// TwinCAT 3 PLC project DrivePLC
// ProgramVersion: 3.1.4020.4
// libraries:
//   Tc2_MC2, * (Beckhoff Automation GmbH)
//   Tc2_MC2_Camming, * (Beckhoff Automation GmbH)
//   Tc2_NC, * (Beckhoff Automation GmbH)
//   Tc2_Standard, * (Beckhoff Automation GmbH)
//   Tc2_System, * (Beckhoff Automation GmbH)
//   Tc3_MC2_AdvancedHoming, * (Beckhoff Automation GmbH)
//   Tc3_Module, * (Beckhoff Automation GmbH)
//   VisuDialogs, * (System)
// project tree:
//   DUTs/ ST_AxisControl.TcDUT, eLimitCoupling.TcDUT, eMcCommand.TcDUT, eRWParameter.TcDUT, ST_MasterAxis.TcDUT, ST_MasterCoupling.TcDUT, ST_SimulateStage.TcDUT
//   / GlobalTextList.TcGTLO, PlcTask.TcTTO, Visualization Manager.TcVMO (not stored)
//   GVLs/ GVL.TcGVL, Limits.TcGVL
//   POUs/ FB_AxisDrive.TcPOU, MAIN.TcPOU
//   VISUs/COMMAND VISUS/ Gearing.TcVIS, Parameters.TcVIS, Homing.TcVIS, AxisSimulation.TcVIS
//   VISUs/ Main.TcVIS
//   VISUs/Panels/ ButtonStates.TcTLO, CommandList.TcTLO, ImagePool.TcIPO (not stored), IO.TcVIS, SlitSet.TcVIS, Visualization.TcVIS
//   VISUs/Panels/Command VISUs/ AxisSimulation.TcVIS, Gearing.TcVIS, Homing.TcVIS, Parameters.TcVIS
// real-time tasks:
//   TASK PlcTask: cycle T#10ms, priority 20, ADS port 350
//   TASK VISU_TASK: cycle T#200000us, priority 30, ADS port 351
// motion (NC):
//   TASK NC-Task 1 SAF: cycle T#2ms, priority 4, ADS port 501
//   TASK NC-Task 1 SVB: cycle T#10ms, priority 8, ADS port 511
//   AXIS NORTH (id 1)
//     General: UnitName=Degree
//     Dynamic: AccelerationMaximum=1500, Acceleration=119.286, Deceleration=119.286, Jerk=424.749
//     Velo: SlowManual=10, FastManual=50, Maximum=50
//     OtherSettings: AllowMotionCmdToSlave=true
//     encoder EncType=1
//     drive DrvType=5
//       Analog: ScaleFactorActTorque=0.1
//       TimeComp: TaskDelayCycles=1
//     controller CtrType=1
//       CtrPara: PriorControlFactor=1
//         Observer: BandWidth=20
//   AXIS SOUTH (id 2)
//     General: UnitName=Degree
//     Dynamic: AccelerationMaximum=1500
//     Velo: SlowManual=10, FastManual=50, Maximum=50
//     OtherSettings: AllowMotionCmdToSlave=true
//     encoder EncType=1
//       EncPara: ScaleFactorNumerator=0.09, Inverse=true
//         SoftEndMaxControl: Range=360
//         Inc: RefSearchInverse=true, RefSyncInverse=false, RefSoftSyncMask=#x0000ffff
//     drive DrvType=5
//       Analog: ScaleFactorActTorque=0.1
//       TimeComp: TaskDelayCycles=1
//     controller CtrType=1
//       CtrPara: PriorControlFactor=1
//         Observer: BandWidth=20
//   AXIS EAST (id 3)
//     General: UnitName=Degree
//     Dynamic: AccelerationMaximum=1500
//     Velo: SlowManual=10, FastManual=50, Maximum=50
//     OtherSettings: AllowMotionCmdToSlave=true
//     encoder EncType=1
//       SoftEndMinControl: Range=-180
//       SoftEndMaxControl: Range=180
//     drive DrvType=5
//       Analog: ScaleFactorActTorque=0.1
//       TimeComp: TaskDelayCycles=1
//     controller CtrType=1
//       CtrPara: PriorControlFactor=1
//         Observer: BandWidth=20
//   AXIS WEST (id 4)
//     Dynamic: AccelerationMaximum=1500
//     Velo: SlowManual=10, FastManual=50, Maximum=50
//     OtherSettings: AllowMotionCmdToSlave=true
//     encoder EncType=1
//       SoftEndMinControl: Range=-180
//       SoftEndMaxControl: Range=180
//     drive DrvType=5
//       Analog: ScaleFactorActTorque=0.1
//       TimeComp: TaskDelayCycles=1
//     controller CtrType=1
//       CtrPara: PriorControlFactor=1
//         Observer: BandWidth=20
//   AXIS VG (id 5)
//     Dynamic: AccelerationMaximum=1500
//     Velo: SlowManual=10, FastManual=50, Maximum=50
//     OtherSettings: AllowMotionCmdToSlave=true
//     encoder EncType=1
//       Inc: RefSoftSyncMask=#x0000ffff
//     drive DrvType=5
//       Analog: ScaleFactorActTorque=0.1
//       TimeComp: TaskDelayCycles=1
//     controller CtrType=1
//       CtrPara: PriorControlFactor=1
//         Observer: BandWidth=20
//   AXIS VC (id 6)
//     Dynamic: AccelerationMaximum=1500
//     Velo: SlowManual=10, FastManual=50, Maximum=50
//     OtherSettings: AllowMotionCmdToSlave=true
//     encoder EncType=1
//     drive DrvType=5
//       Analog: ScaleFactorActTorque=0.1
//       TimeComp: TaskDelayCycles=1
//     controller CtrType=1
//       CtrPara: PriorControlFactor=1
//         Observer: BandWidth=20
//   AXIS HG (id 7)
//     Dynamic: AccelerationMaximum=1500
//     Velo: SlowManual=10, FastManual=50, Maximum=50
//     OtherSettings: AllowMotionCmdToSlave=true
//     encoder EncType=1
//     drive DrvType=5
//       Analog: ScaleFactorActTorque=0.1
//       TimeComp: TaskDelayCycles=1
//     controller CtrType=1
//       CtrPara: PriorControlFactor=1
//         Observer: BandWidth=20
//   AXIS HC (id 8)
//     Dynamic: AccelerationMaximum=1500
//     Velo: SlowManual=10, FastManual=50, Maximum=50
//     OtherSettings: AllowMotionCmdToSlave=true
//     encoder EncType=1
//     drive DrvType=5
//       Analog: ScaleFactorActTorque=0.1
//       TimeComp: TaskDelayCycles=1
//     controller CtrType=1
//       CtrPara: PriorControlFactor=1
//         Observer: BandWidth=20
// variable links:
//   DrivePLC Instance <-> NC-Task 1 SAF/Axes/EAST
//     PlcTask Inputs/GVL.axes[3].Axis.NcToPlc <-> Outputs/ToPlc
//     PlcTask Outputs/GVL.axes[3].Axis.PlcToNc <-> Inputs/FromPlc
//   DrivePLC Instance <-> NC-Task 1 SAF/Axes/HC
//     PlcTask Inputs/GVL.axes[8].Axis.NcToPlc <-> Outputs/ToPlc
//     PlcTask Outputs/GVL.axes[8].Axis.PlcToNc <-> Inputs/FromPlc
//   DrivePLC Instance <-> NC-Task 1 SAF/Axes/HG
//     PlcTask Inputs/GVL.axes[7].Axis.NcToPlc <-> Outputs/ToPlc
//     PlcTask Outputs/GVL.axes[7].Axis.PlcToNc <-> Inputs/FromPlc
//   DrivePLC Instance <-> NC-Task 1 SAF/Axes/NORTH
//     PlcTask Inputs/GVL.axes[1].Axis.NcToPlc <-> Outputs/ToPlc
//     PlcTask Outputs/GVL.axes[1].Axis.PlcToNc <-> Inputs/FromPlc
//   DrivePLC Instance <-> NC-Task 1 SAF/Axes/SOUTH
//     PlcTask Inputs/GVL.axes[2].Axis.NcToPlc <-> Outputs/ToPlc
//     PlcTask Outputs/GVL.axes[2].Axis.PlcToNc <-> Inputs/FromPlc
//   DrivePLC Instance <-> NC-Task 1 SAF/Axes/VC
//     PlcTask Inputs/GVL.axes[6].Axis.NcToPlc <-> Outputs/ToPlc
//     PlcTask Outputs/GVL.axes[6].Axis.PlcToNc <-> Inputs/FromPlc
//   DrivePLC Instance <-> NC-Task 1 SAF/Axes/VG
//     PlcTask Inputs/GVL.axes[5].Axis.NcToPlc <-> Outputs/ToPlc
//     PlcTask Outputs/GVL.axes[5].Axis.PlcToNc <-> Inputs/FromPlc
//   DrivePLC Instance <-> NC-Task 1 SAF/Axes/WEST
//     PlcTask Inputs/GVL.axes[4].Axis.NcToPlc <-> Outputs/ToPlc
//     PlcTask Outputs/GVL.axes[4].Axis.PlcToNc <-> Inputs/FromPlc

CONFIGURATION DrivePLC
    RESOURCE PLC ON TwinCAT3
        TASK PlcTask(INTERVAL := T#10ms, PRIORITY := 20);
        PROGRAM MAIN WITH PlcTask : MAIN;
    END_RESOURCE
END_CONFIGURATION

// ---- DUTs/ST_AxisControl.TcDUT
TYPE ST_AxisControl :
STRUCT
	//OPC UA functionality not implemented yet
	(*For a list of parameters required to operate each motion control funciton block
	see the DUT eMcCommand*)
	
	bExecute			:	BOOL;			//Rising edge to execute command
	bReset				:	BOOL;			//Reset axis signal, must be combined with other signals
	eCommand			:	eMcCommand;		//Motion command for axis
	bEnable				: 	BOOL;			//Controller enable
	fOverride			:	LREAL;			//Controller override %
	fVelocity			:	LREAL;			//Velocity must be specified, no default used
	fAcceleration		:	LREAL;			//Not all FBs use, need to change this, 0 is NC default
	fDeceleration		:	LREAL;			//Not all FBs use, need to change this, 0 is NC default
	fDistance			:	LREAL;			//Used for relative positioning
	fPosition			:	LREAL;			//Used for absolute positioning	
	bJogForward			:	BOOL;			//Jog forward
	bJogBackward		:	BOOL;			//Jog backward
	
	bInput				:	BOOL;			//Generic input that is utilised to control some functionality
	
	bSoftLimPosEn		:	BOOL;			//Enable/disable positive direction software limit
	bSoftLimNegEn		:	BOOL;			//Enable/disable negative direction software limit
	bPosLagEn			:	BOOL;			//Enable/disable position lag
	
	//Gearing parameters
	masterAxis			:	UINT:=1;						//Axes[ ] index for master		- GearIn
	fGearRatioNum		:	LREAL;							//GearIn ratio numerator
	iGearRatioDen		:	UINT;							//GearIn ratio denominator
	masterAxes			:	ARRAY[1..4] OF ST_MasterAxis;	//ST to hold index and ratio for masters 	- GearInMultiMaster
	
	//NC Parameters	
	iParameterIndex		:	INT;					//Index for checking parameters
	fParameterValue		:	LREAL;					//Holder for assigning new values
	fParameters			:	ARRAY [1..17] OF LREAL;	//Array to hold NC parameters
	
	//MISC
	sAxisName			:	STRING;					//User set name string for axis
	sAxisDesc			:	STRING;					//User set description string for axis
	
	//Outputs
	bFwEnabled			:	BOOL;					//Positive movement of axis is enabled/disabled
	bBwEnabled			:	BOOL;					//Negative movement of axis is enabled/disabled
	bAxisReady			:	BOOL;					//Output of McPower block	
	bError				:	BOOL;					//Motion function block has produced error (NC drive not necessarily in error state)
	iErrorID			:	UDINT;					//Motion function block errorID				
	bBusy				:	BOOL;					//Axis busy
	bMoving				:	BOOL;					//Axis moving					
	bDone				:	BOOL;					//Last function block executed successfully			
	
	iAxisState			:	UINT;					//PLC Open NC statemachine, int assigned to individual NC bool state outputs
	(*	100 - Disabled
		200 - Standstill
		300 - Homing
		400 - Discrete Motion
		500 - Synchronized Motion
		600 - Continuous Motion
		700 - Stopping
		999 - Error
	*)
	
	buffer				:	MC_BufferMode;							//Placeholder - Not currently used
	
	//Homing
	fHomeVelocity		:	LREAL	:=1;							//Homing routine velocity 							- initialised for testing purposes
	fHomeTorque			:	LREAL;									//Homing torque limit (not all drives support this)
	fHomePosition		:	LREAL;									//Position set at NC when homing step finished
	fHomeDistance		:	LREAL;									//Relative distance to move after homing
	tHomeTimeLimit		:	TIME:=T#60S;							//Homing timeout limit, FB errors is exceeded 		- initialised for testing purposes
	fHomeDistanceLimit	:	LREAL:=2000;							//Homing distance limit, FB errors if exceeded 		- initialised for testing purposes
	
	MCHomeDirection		:	MC_Home_Direction:=	mcSwitchPositive;	//init for testing purposes
	(*	Direction to begin homing. Not all are compatible with every advanced homing step
		mcPositiveDirection	-	always start positive
		mcNegativeDirection	-	always start negative
		mcSwitchPositive	-	start positive unless already on the switch
		mcSwitchNegative	-	start negative unless already on the switch
		
	*)
	

	MCSwitchMode		:	MC_Switch_Mode:= mcRisingEdge;			//init for testing purposes
	(* Switch detection behaviour, I am not entirely convinced these are all working as they are meant to, further work required. Not all detection methods work with every 
	step either so they have to be updated.
		mcOn
		mcOff
		mcRisingEdge
		mcFallingEdge
		mcEdgeSwitchPositive
		mcEdgeSwitchNegative
		mcRisingEdgeInverse
		mcFallingEdgeInverse	
	*)

	MCSignalRef			:	MC_Ref_Signal_Ref;						//In structure for testing purposes so I can simulate level of signal without hardware
	(*Further investigation required on how exactly this MCSignalRef works, it seems to contain signalsource, touch probe and level signals,
	my current understanding is that with physical hardware connected the MCSignalRef signal source should default to the NC hardware so nothing has to be linked
	for the encoder index, however the source may need to be changed for the absSwitch homing which would just require an additional line of code in the driveFB step command
	I also do not have any bool available for linking an absolute switch to an axis at the moment

		SignalSource : E_SignalSource := SignalSource_Default;
		TouchProbe : E_TouchProbe := PlcEvent;
		Level : BOOL;

	*)

	// Data for EPICS from the axis ref
	fActPosition   			: LREAL;
	fActVelocity  		 	: LREAL;
	bNegativeDirection 		: BOOL;
	bPositiveDirection		: BOOL;
	bCalibrated 			: BOOL;
	
	Axis				:	AXIS_REF;		(*~ (OPC: 0 : available for OPC-clients) *)

END_STRUCT
END_TYPE

// ---- DUTs/eLimitCoupling.TcDUT
{attribute 'qualified_only'}
{attribute 'strict'}
(*
	Structure used to couple limit switches of slaves to master axes
*)
TYPE eLimitCoupling :
(
	None,
	FwSw,
	BwSw
);
END_TYPE

// ---- DUTs/eMcCommand.TcDUT
{attribute 'qualified_only'}
{attribute 'strict'}
TYPE eMcCommand :
(
	(*
		Only those with listed inputs have been implemented, the rest are placeholders to be added 
		To utilise a listed command you must give the ST_AxisControl the listed inputs, the drive function block will latch on a command until it is complete or errors 
		and the bExecute signal will be automatically set FALSE on every cycle
	*)
	
	Idle,					//Internal idle command, 	Inputs	:	NONE
	Reset,					//Reset NC axis,			Inputs	:	bReset
	ReadAxisError,
	WriteParameter,			//Write to NC parameters,	Inputs	:	bExecute	iParameterIndex		fParameterValue
	WriteBoolParameter,		//Write to NC parameters,	Inputs	:	bExecute	iParameterIndex		bInput

	ReadActualPosition,
	ReadActualVelocity,

	
	SetPosition,			//Set NC axis position,		Inputs	:	bExecute	fPosition			
	SetOverride,
	TouchProbe,
	
	AbortTrigger,
	AbortSuperposition,
	CamTableSelect,
	
	Home,
	Jog,					//Jog the axis,				Inputs	:	bJogForward		bJogBackward
	Stop,					//Stop axis motion,			Inputs	:	bExecute	fDeceleration
	Halt,
	MoveAbsolute,			//Absolute move,			Inputs	:	bExecute	fPosition	fVelocity	fAcceleration	fDeceleration
	MoveRelative,			//Relative move,			Inputs	:	bExecute	fDistance	fVelocity	fAcceleration	fDeceleration
	MoveAdditive,
	MoveSuperimposed,
	MoveVelocity,			//Velocity move,			Inputs	:	bExecute	fVelocity	fAcceleration	fDeceleration
	MoveContinuousAbs,
	MoveContinuousRel,
	MoveModulo,
	
	GearIn,					//Single master gear in,	Inputs	:	bExecute	fGearRatioNum	iGearRatioDen	masterAxis
	GearInDyn,
	GearInMultiMaster,		//Multi master gear in,		Inputs	:	bExecute	fGearRatio1		fGearRatio2		fGearRatio3		fGearRatio4		masterAxis1		masterAxis2		masterAxis3		masterAxis4
	GearOut,				//Release gearing,			Inputs	:	bExecute	
	HaltPhasing,
	PhasingAbsolute,
	PhasingRelative,
	CamIn,
	CamOut,
	CamScaling,
	CamAdd,
	CamExchange,
	CamInV2,
	CamRemove,
	CamScalingV2,
	
	//HOMING		Those marked with * have had values initialised and don't need to be input (but can be)
	HomeFinish,				//Finish homing routin,		Inputs	:	bExecute	fHomeDistance	fHomeVelocity
	HomeDirect,
	HomeAbort,
	HomeStepAbsoluteSwitch,	//Homing step,				Inputs	:	bExecute	MCHomeDirection*	mcSwitchMode*	mcSignalRef*	fHomeVelocity*	fHomeTorque		fHomePosition	tHomeTimeLimit*		fHomeDistanceLimit*		buffer*
	HomeStepBlock,
	HomeStepBlockLagBased,
	HomeStepLimitSwitch,
	HomeStepReferencePulse
	
);
END_TYPE

// ---- DUTs/eRWParameter.TcDUT
{attribute 'qualified_only'}
{attribute 'strict'}
TYPE eRWParameter :
(
	CommandedPosition 		:= 1,	//REAL		R	- Commanded position
	SWLimitPos				:= 2,	//REAL		R/W	- Positive Software limit switch position
	SWLimitNeg				:= 3,	//REAL		R/W	- Negative Software limit switch position
	EnableLimitPos			:= 4,	//BOOL		R/W	- Enable positive software limit switch
	EnableLimitNeg			:= 5, 	//BOOL		R/W	- Enable negative software limit switch
	EnablePosLagMonitoring	:= 6,	//BOOL		R/W	- Enable monitoring of position lag
	MaxPositionLag			:= 7,	//REAL		R/W	- Maximal position lag
	MaxVelocitySystem		:= 8,	//REAL		R	- Maximal allowed velocity of the axis in the motion system
	MaxVelocityAppl			:= 9,	//REAL		R/W	- Maximal allowed velocity of the axis in the application
	ActualVelocity			:= 10,	//REAL		R	- Actual velocity
	CommandedVelocity		:= 11,	//REAL		R	- Commanded velocity
	MaxAccelerationSystem	:= 12,	//REAL		R	- Maximal allowed acceleration of the axis in the motion system
	MaxAccelerationAppl		:= 13,	//REAL		R/W	- Maximal allowed acceleration of the axis in the application
	MaxDecelerationSystem	:= 14,	//REAL		R	- Maximal allowed deceleration of the axis in the motion system
	MaxDecelerationAppl		:= 15,	//REAL		R/W	- Maximal allowed deceleration of the axis in the application
	MaxJerkSystem			:= 16,	//REAL		R	- Maximum allowed jerk of the axis in the motion system
	MaxJerkAppl				:= 17	//REAL		R/W	- Maximum allowed jerk of the axis in the application
);
END_TYPE

// ---- DUTs/ST_MasterAxis.TcDUT
(*
	Strucure to hold master axes information for the GearInMultiMaster command
*)
TYPE ST_MasterAxis :
STRUCT
	i		:	UINT:=1;	//Master axis index
	ratio	:	LREAL;		//Gearing Ratio
END_STRUCT
END_TYPE

// ---- DUTs/ST_MasterCoupling.TcDUT
(*
	Structure for storing link information to enable limit passing from slaves to masters
*)
TYPE ST_MasterCoupling :
STRUCT
	iMasterAxis		:	UINT	:=1;		//Must be initialised to 1 as no 0 index on arrays
	eLimitType		:	eLimitCoupling;
END_STRUCT
END_TYPE

// ---- DUTs/ST_SimulateStage.TcDUT
TYPE ST_SimulateStage :
STRUCT
	//High and low limits for simulating axes
	fHighLim	:	LREAL	:=10;
	fLowLim		:	LREAL	:=-10;
	fHighAbs	:	LREAL	:=1;
	fLowAbs		:	LREAL	:=-1;
	absSw		:	BOOL;
END_STRUCT
END_TYPE

// ---- GVLs/GVL.TcGVL
{attribute 'qualified_only'}
VAR_GLOBAL
	iAxis		:	UINT; //Indexing variable for exposing which axis currently being run though drive function block
	axes			:	ARRAY [1..GVL.axisNumMax] OF ST_AxisControl;		(*~ (OPC: 1 : available for OPC-clients) 
	    																		(OPC_PROP[0005]: 3 : OPC_PROP_RIGHTS, here read/write) *)
//HMI Parameters	-	These can hopefully be removed on upgrading to the new HMI tool
	SwLimitPos	:	LREAL;
	SwLimitNeg	:	LREAL;
	MaxPositionLag	:	LREAL;
	MaxVelocityAppl	:	LREAL;
	MaxAccelerationAppl	:	LREAL;
	MaxDecelerationAppl	:	LREAL;
	MaxJerkAppl			:	LREAL;
	
END_VAR
VAR_GLOBAL CONSTANT
	axisNumMax	:	UINT:=8;
	axisCoupleMax	:	UINT:=4;
END_VAR

// ---- GVLs/Limits.TcGVL
{attribute 'qualified_only'}
VAR_GLOBAL
	FwLimit				AT	%I*	: ARRAY[1..GVL.axisNumMax] OF BOOL;		(*~ (OPC: 1 : available for OPC-clients) 
	    																(OPC_PROP[0005]: 3 : OPC_PROP_RIGHTS, here read/write) *)
																		//Forward limit hardware link (opc available for testing)
																		
	BwLimit				AT  %I*	: ARRAY[1..GVL.axisNumMax] OF BOOL;		(*~ (OPC: 1 : available for OPC-clients) 
	    																(OPC_PROP[0005]: 3 : OPC_PROP_RIGHTS, here read/write) *)
																		//Backward limit hardware link (opc available for testing)
	
	coupledFwLimit		: ARRAY [1..GVL.axisNumMax] OF ARRAY [1..5] OF ST_MasterCoupling;	//Store for slave/master linking
	coupledBwLimit		: ARRAY [1..GVL.axisNumMax] OF ARRAY [1..5] OF ST_MasterCoupling;	//Store for slave/master linking

END_VAR

// ---- POUs/MAIN.TcPOU
PROGRAM MAIN
VAR
	//Simulate virtual axes
	simulated		:	ARRAY [1..GVL.axisNumMax] OF ST_SimulateStage;
	bSimulate		:	ARRAY [1..GVL.axisNumMax] OF BOOL;	//Do we want to simulate?
	
	drives			:	ARRAY [1..GVL.axisNumMax] OF FB_AxisDrive;	
	
	bDisableMC		:	BOOL; 		//boolean control if true the motion control application specific code is disabled - dumb box
	iState			:	UINT;		//state machine index

	(*
		Outputs that are set in the hmi and wired to power axis limit switches. Currently not configred as part of the programme
		Will be added to ST_AxisControl in future
	*)
	limitEnable1	AT %Q*	: BOOL;
	limitEnable2	AT %Q*	: BOOL;	
	
	i: UINT;		//General indexing value for FOR loops	
	
	//HMI VARIABLES	
	hmiAxisSelect	:	UINT:=1;

END_VAR

AXES();
PROG();
SIMULATE();

ACTION AXES:
FOR GVL.iAxis:=1 TO GVL.axisNumMax DO
	drives[GVL.iAxis](AxisController:=GVL.axes[GVL.iAxis]);
END_FOR
END_ACTION

(*
	Scans through axes (from low to high) checking "done" status
*)
METHOD CheckDone : BOOL
VAR_INPUT
	iLow	:	UINT;		//lowest index to check
	iHigh	:	UINT;		//highest index to check
END_VAR

VAR
	i		:	UINT;
END_VAR
CheckDone:=TRUE;
FOR i:=iLow TO iHigh BY 1 DO
	CheckDone:= CheckDone AND GVL.axes[i].bDone;
END_FOR
END_METHOD

(*
	Gear out an axis
*)
METHOD GearOut : BOOL
VAR_INPUT
	i	:	UINT;	//Axis index to gear out
END_VAR
GVL.axes[i].eCommand:=eMcCommand.GearOut;
GVL.axes[i].bExecute:=TRUE;
END_METHOD

(*
	Power up a single axis of index i
*)
METHOD PowerUp : BOOL
VAR_INPUT
	i	:	UINT;
END_VAR
GVL.axes[i].bEnable:=TRUE;
GVL.axes[i].fOverride:=100;
Limits.FwLimit[i]:=TRUE;	//Set high as I have no hardware linked
Limits.BwLimit[i]:=TRUE;	//Set high as I have no hardware linked
END_METHOD

ACTION PROG:
CASE iState OF
	0:	//CHECK AXIS ID's are correct. Gearing limits currently requires the assigned array index of an axis to match the NC ID.
		//May be possible to negate this by changing axes to GVLs so that they can be seen within the drives function - CASE 0 NO LONGER REQ
		iState:=1;
		FOR i:=1 TO GVL.axisNumMax BY 1 DO
			IF GVL.axes[i].Axis.NcToPlc.AxisId <> i THEN
				iState:=999;
			END_IF
		END_FOR
		
	1:	//Gear out all axes to begin
		FOR i:=1 TO 8 BY 1 DO
			GearOut(i:=i);
		END_FOR
		iState:= 2;
	2:	//Wait for gear out
		IF CheckDone(iLow:=1, iHigh:=8) THEN
			iState:=3;
		END_IF
	3:	//Power up axes (and set limits true as no hardware connected)
		FOR i:=1 TO 8 BY 1 DO
			PowerUp(i:=i);
		END_FOR
		iState:= 10;
		
	10:	//Set position of virtual gap axes based on position. In reality we would do some homing sequence of blades first then set the position
		SlitPositions(North:=1,South:=2,East:=3,West:=4,VG:=5,VC:=6,HG:=7,HC:=8);
		iState:=11;
		
	11:	//Wait for position set
		IF CheckDone(iLow:=5,iHigh:=8) THEN
			iState:=12;
		END_IF		
		
	12:	//GEAR IN SLIT GAP AND CENTRE
		SlitSetup(North:=1,South:=2,East:=3,West:=4,VG:=5,VC:=6,HG:=7,HC:=8);
		iState:=13;
	
	13:	//WAIT FOR DONE
		IF CheckDone(iLow:=1, iHigh:=4) THEN
			iState:=14;
		END_IF	

	14: //ALL SETUP!	
			IF bDisableMC THEN
				iState:=50;
			END_IF
	
	50:
		FOR i:=1 TO 8 BY 1 DO
			GearOut(i:=i);
		END_FOR
		iState:=51;
	51:
		IF CheckDone(iLow:=1, iHigh:=8) THEN
			iState:=100;
		END_IF					
			
	100:	//DO NOTHING


		
		IF NOT bDisableMC THEN
			iState:=1;
		END_IF

		
	
	999: //ERROR
		//INOP STATE	
END_CASE
END_ACTION

ACTION SIMULATE:
(*
Simulate axes if bool set TRUE
*)
FOR i:=1 TO GVL.axisNumMax BY 1 DO
	IF bSimulate[i] THEN
		simulateStage(position:=GVL.axes[i].Axis.NcToPlc.ActPos, iAxis:=i, simulated:=simulated[i]);
		GVL.axes[i].MCSignalRef.Level:=simulated[i].absSw;
	END_IF
END_FOR
END_ACTION

(*
	Basic virtual axis simulation.
	Will trigger limit switches beyond set points
	Will trigger absolute switch between given set points
*)
METHOD simulateStage : BOOL
VAR_INPUT
	position	:	LREAL;		//Axis current position
	iAxis		:	UINT;		//Axis index
END_VAR
VAR_IN_OUT
	simulated	:	ST_SimulateStage;	//Struct to hold simulation parameters
END_VAR
Limits.FwLimit[iAxis]:= position < simulated.fHighLim;
Limits.BwLimit[iAxis]:= position > simulated.fLowLim;

simulated.absSw:= (position < simulated.fHighAbs) AND (position > simulated.fLowAbs);
END_METHOD

(*
	Calculate gap positions of a slit set given N/S/E/W blades
*)
METHOD SlitPositions : BOOL
VAR_INPUT
	North	:	UINT;	//North blade index
	South	:	UINT;	//South blade index
	East	:	UINT;	//East blade index
	West	:	UINT;	//West blade index
	VG		:	UINT;	//Vertical gap size index
	VC		:	UINT;	//Vertical gap centre index
	HG		:	UINT;	//Horizontal gap size index
	HC		:	UINT;	//Horizontal gap centre index
END_VAR
GVL.axes[VG].eCommand:=eMcCommand.SetPosition;
GVL.axes[VG].fPosition:=GVL.axes[North].Axis.NcToPlc.ActPos-GVL.axes[South].Axis.NcToPlc.ActPos;
GVL.axes[VG].bExecute:=TRUE;

GVL.axes[VC].eCommand:=eMcCommand.SetPosition;
GVL.axes[VC].fPosition:=(GVL.axes[North].Axis.NcToPlc.ActPos+GVL.axes[South].Axis.NcToPlc.ActPos)/2;
GVL.axes[VC].bExecute:=TRUE;

GVL.axes[HG].eCommand:=eMcCommand.SetPosition;
GVL.axes[HG].fPosition:=GVL.axes[East].Axis.NcToPlc.ActPos-GVL.axes[West].Axis.NcToPlc.ActPos;
GVL.axes[HG].bExecute:=TRUE;

GVL.axes[HC].eCommand:=eMcCommand.SetPosition;
GVL.axes[HC].fPosition:=(GVL.axes[East].Axis.NcToPlc.ActPos+GVL.axes[West].Axis.NcToPlc.ActPos)/2;
GVL.axes[HC].bExecute:=TRUE;
END_METHOD

(*
	Gear in blades to gaps for a slit set
*)
METHOD SlitSetup : BOOL
VAR_INPUT
	North	:	UINT;
	South	:	UINT;
	East	:	UINT;
	West	:	UINT;
	VG		:	UINT;
	VC		:	UINT;
	HG		:	UINT;
	HC		:	UINT;
END_VAR
GVL.axes[North].eCommand:= eMcCommand.GearInMultiMaster;
GVL.axes[North].bExecute:=TRUE;
GVL.axes[NORTH].masterAxes[1].i:=VG;
GVL.axes[NORTH].masterAxes[2].i:=VC;
GVL.axes[NORTH].masterAxes[1].ratio:=0.5;
GVL.axes[NORTH].masterAxes[2].ratio:=1;

GVL.axes[South].eCommand:= eMcCommand.GearInMultiMaster;
GVL.axes[South].bExecute:=TRUE;
GVL.axes[South].masterAxes[1].i:=VG;
GVL.axes[South].masterAxes[2].i:=VC;
GVL.axes[South].masterAxes[1].ratio:=-0.5;
GVL.axes[South].masterAxes[2].ratio:=1;

GVL.axes[West].eCommand:= eMcCommand.GearInMultiMaster;
GVL.axes[West].bExecute:=TRUE;
GVL.axes[West].masterAxes[1].i:=HG;
GVL.axes[West].masterAxes[2].i:=HC;
GVL.axes[West].masterAxes[1].ratio:=-0.5;
GVL.axes[West].masterAxes[2].ratio:=1;


GVL.axes[East].eCommand:= eMcCommand.GearInMultiMaster;
GVL.axes[East].bExecute:=TRUE;
GVL.axes[East].masterAxes[1].i:=HG;
GVL.axes[East].masterAxes[2].i:=HC;
GVL.axes[East].masterAxes[1].ratio:=0.5;
GVL.axes[East].masterAxes[2].ratio:=1;
END_METHOD

END_PROGRAM

// ---- POUs/FB_AxisDrive.TcPOU
(*
	Function for motion control of single axis.
	Provides an interface to PLC Open motion control blocks.
	Controls linking of limit switches from slave to master axes.
*)
FUNCTION_BLOCK FB_AxisDrive
VAR_INPUT
END_VAR
VAR_IN_OUT
	AxisController		:	ST_AxisControl;
END_VAR
VAR_OUTPUT
END_VAR
VAR
	eCommandLatched		:	eMcCommand;		//Internally latched command signal, new commands cannot be issued until existing commands have completed.
	doneLatch	:	SR;						//Used to set done signal in AxisController DUT
	bDone		:	BOOL;					//Interal done flag which will be used for latching on an external done located in AxisController DUT
	iParam		:	INT:=1;					//index of NC parameters FBs, no 0 index on array so initialised to 1
	iIndex		:	UINT;					//index value used for limit coupling
	iMasterIndex		:	UINT;			//index value used for limit coupling
	
	//Boolean to store EnableFw and EnableBw of MCPower FB
	FwLimitsEnabled	:	BOOL;	
	BWLimitsEnabled	:	BOOL;
	
	mcDirection	:	MC_Direction;			//Direction control required in function blocks

(*
Motion Function blocks taken from the PLC OPEN standard as defined by PLC Open Standard
Function blocks commented out are yet to be added but the intention is to add these.
Those listed as //NOT IMPLEMENTED have come from the standard but Beckhoff do not support, 
these have been added just as a placeholder for future support.
*)
	//Not Implemented
	//MCReadDigitalInput		:	MC_ReadDigitalInput;			//NOT IMPLEMENTED		
	//MCReadDigitalOutput		:	MC_ReadDigitalOutput;			//NOT IMPLEMENTED	
	//MCWriteDigitalOutput		:	MC_WriteDigitalOutput;			//NOT IMPLEMENTED
	//MCReadActualTorque		:	MC_ReadActualTorque;			//NOT IMPLEMENTED	
	//MCReadAxisInfo			:	MC_ReadAxisInfo;				//NOT IMPLEMENTED	
	//MCReadMotionState			:	MC_ReadMotionState;				//NOT IMPLEMENTED
	//MCDigitalCamSwitch		:	MC_DigitalCamSwitch;			//NOT IMPLEMENTED
	//MCTorqueControl			:	MC_TorqueControl;				//NOT IMPLEMENTED		
	//MCPositionProfile			:	MC_PositionProfile;				//NOT IMPLEMENTED		
	//MCVelocityProfile			:	MC_VelocityProfile;				//NOT IMPLEMENTED		
	//MCAccelerationProfile		:	MC_AccelerationProfile;			//NOT IMPLEMENTED
	
	
	(* Administrative Function Blocks *)                                                                     
	MCReset						:	MC_Reset;											
	MCPower						:	MC_Power;										
	//MCReadStatus				:	MC_ReadStatus;					//Same as Axis.ReadStatus();						
	//MCReadAxisError			:	MC_ReadAxisError;									
	MCReadParameter				:	MC_ReadParameter;														
	MCWriteParameter			:	MC_WriteParameter;										
	MCWriteBoolParameter		:	MC_WriteBoolParameter;								
		
	//MCReadActualPosition		:	MC_ReadActualPosition;								
	//MCReadActualVelocity		:	MC_ReadActualVelocity;								
		
	MCSetPosition				:	MC_SetPosition;										
	//MCSetOverride				:	MC_SetOverride;										
	//MCTouchProbe				:	MC_TouchProbe;										
		
	//MCAbortTrigger			:	MC_AbortTrigger;									
	//MCAbortSuperposition		:	MC_AbortSuperposition;			//Listed as HaltSuperimposed in PLC Open standard	
	//MCCamTableSelect			:	MC_CamTableSelect;									
	
	(* Motion Function Blocks *)
	//MCHome					:	MC_Home;											
	MCJog						:	MC_Jog;												
	MCStop						:	MC_Stop;											
	//MCHalt					:	MC_Halt;											
	MCMoveAbsolute				:	MC_MoveAbsolute;									
	MCMoveRelative				:	MC_MoveRelative;									
	//MCMoveAdditive			:	MC_MoveAdditive;									
	//MCMoveSuperimposed		:	MC_MoveSuperimposed;								
	MCMoveVelocity				:	MC_MoveVelocity;									
	//MCMoveContinuousAbsolute	:	MC_MoveContinuousAbsolute;						
	//MCMoveContinuousRelative	:	MC_MoveContinuousRelative;						
	//MCMoveModulo				:	MC_MoveModulo;										
	
	(* Synchronised Motion Function Blocks *)		
	MCGearIn					:	MC_GearIn;											
	//MCGearInDyn				:	MC_GearInDyn;										
	MCGearInMultiMaster			:	MC_GearInMultiMaster;								
	MCGearOut					:	MC_GearOut;												                                                                                    
	//MCHaltPhasing				:	MC_HaltPhasing;										
	//MCPhasingAbsolute			:	MC_PhasingAbsolute;									
	//MCPhasingRelative			:	MC_PhasingRelative;										                                                                                                                                                 
	//MCCamIn					:	MC_CamIn;											
	//MCCamOut					:	MC_CamOut;											
	//MCCamScaling				:	MC_CamScaling;										                                                      
	//MCCamAdd					:	MC_CamAdd;											
	//MCCamExchange				:	MC_CamExchange;										
	//MCCamInV2					:	MC_CamIn_V2;		//REQUIRED FOR MULTICAMMING 	
	//MCCamRemove				:	MC_CamRemove;										
	//MCCamScalingV2			:	MC_CamScaling_V2;									

	(* Advanced Homing Steps and Finishing Moves *)
	MCFinishHoming			:	MC_FinishHoming;
	//MCHomeDirect			:	MC_HomeDirect;
	//MCAbortHoming			:	MC_AbortHoming;
	MCStepAbsoluteSwitch	:	MC_StepAbsoluteSwitch;
	//MCStepBlock			:	MC_StepBlock;
	//MCStepBlockLagBased	:	MC_StepBlockLagBased;
	//MCStepLimitSwitch		:	MC_StepLimitSwitch;
	//MCStepReferencePulse	:	MC_StepReferencePulse;
	
	
	(* Additional variable structures required for Advanced Homing *)
	//MCSignalRef			:	MC_Ref_Signal_Ref;
	StOptions				:	ST_Home_Options;
	StOptions2				:	ST_Home_Options2;
	StOptions3				:	ST_Home_Options3;
	StOptions4				:	ST_Home_Options4;
	MCHomingParameter		:	MC_HomingParameter;		//Must be passed between homing steps.		
							
END_VAR

AxisController.Axis.ReadStatus();

// Pass data through for EPICS to read
AxisController.fActPosition:= AxisController.Axis.NcToPlc.ActPos;
AxisController.fActVelocity:= AxisController.Axis.NcToPlc.ActVelo;
AxisController.bNegativeDirection:= AxisController.Axis.Status.NegativeDirection;
AxisController.bPositiveDirection:= AxisController.Axis.Status.PositiveDirection;
AxisController.bCalibrated:= AxisController.Axis.Status.Homed;

//////////////////////////////////////////////////////////////////////
//     _   __  _____ ____    ____ _____  _  _____ _____ ____  		//
//    / \  \ \/ |_ _/ ___|  / ___|_   _|/ \|_   _| ____/ ___| 		//
//   / _ \  \  / | |\___ \  \___ \ | | / _ \ | | |  _| \___ \ 		//
//  / ___ \ /  \ | | ___) |  ___) || |/ ___ \| | | |___ ___) |		//
// /_/   \_/_/\_|___|____/  |____/ |_/_/   \_|_| |_____|____/ 		//
// 																	//
//////////////////////////////////////////////////////////////////////
                                                            
//Numerical representation for axis states - may use later for buffering functions.
IF AxisController.AXIS.Status.Disabled THEN
	AxisController.iAxisState:=		100;
ELSIF AxisController.AXIS.Status.StandStill THEN
	AxisController.iAxisState:=		200;
ELSIF AxisController.AXIS.Status.Homing	THEN
	AxisController.iAxisState:= 	300;
ELSIF AxisController.AXIS.Status.DiscreteMotion	THEN
	AxisController.iAxisState:=		400;
ELSIF AxisController.AXIS.Status.SynchronizedMotion	THEN
	AxisController.iAxisState:=		500;
ELSIF AxisController.AXIS.Status.ContinuousMotion	THEN
	AxisController.iAxisState:=		600;
ELSIF AxisController.AXIS.Status.Stopping	THEN
	AxisController.iAxisState:= 	700;	
ELSIF AxisController.AXIS.Status.Error THEN
	AxisController.iAxisState:=		999;	
ELSE
	AxisController.iAxisState:=		0;
END_IF

//////////////////////////////////////////////////////////////////////////////////////////
//  _     ___ __  __ ___ _____   ______        _____ _____ ____ _   _ _____ ____  		//
// | |   |_ _|  \/  |_ _|_   _| / ___\ \      / |_ _|_   _/ ___| | | | ____/ ___| 		//
// | |    | || |\/| || |  | |   \___ \\ \ /\ / / | |  | || |   | |_| |  _| \___ \ 		//
// | |___ | || |  | || |  | |    ___) |\ V  V /  | |  | || |___|  _  | |___ ___) |		//
// |_____|___|_|  |_|___| |_|   |____/  \_/\_/  |___| |_| \____|_| |_|_____|____/		//
//																						//
//////////////////////////////////////////////////////////////////////////////////////////

//Initialise Foward and Backward limits to the hardware limit switches for this axis
FwLimitsEnabled :=Limits.FwLimit[GVL.iAxis];
BwLimitsEnabled :=Limits.BwLimit[GVL.iAxis];

(*
Cycle through Limits.coupledFwLimit and Limits.coupledBwLimit.
Looking to see if any axes have the current axis (GVL.iAxis) listed as a master.
If this axis is listed as a master, check the hardware limits of that slave.
Gear ratio determines whether we are looking for a Forward or a Backward limit on the slave axis. 
If the limit switch is disabled, disable motion for this axis.
*)
FOR iIndex:=1 TO GVL.axisNumMax DO
	FOR iMasterIndex:=1 TO 5 DO
		//If listed as a master
		IF Limits.coupledFwLimit[iIndex][iMasterIndex].iMasterAxis = GVL.iAxis THEN
			//If forward limit linked to forward of slave, check forward limit of slave
			IF Limits.coupledFwLimit[iIndex][iMasterIndex].eLimitType=eLimitCoupling.FwSw AND NOT Limits.FwLimit[iIndex] THEN
				FwLimitsEnabled:=FALSE;
			END_IF
			//If forward limit linked to backwardof slave, check forward limit of slave
			IF Limits.coupledFwLimit[iIndex][iMasterIndex].eLimitType=eLimitCoupling.BwSw AND NOT Limits.BwLimit[iIndex] THEN
				FwLimitsEnabled:=FALSE;
			END_IF
			//If backward limit linked to forward of slave, check forward limit of slave
			IF Limits.coupledBwLimit[iIndex][iMasterIndex].eLimitType=eLimitCoupling.FwSw AND NOT Limits.FwLimit[iIndex] THEN
				BwLimitsEnabled:=FALSE;
			END_IF
			//If backward limit linked to backward of slave, check backward limit of slave
			IF Limits.coupledBwLimit[iIndex][iMasterIndex].eLimitType=eLimitCoupling.BwSw AND NOT Limits.BwLimit[iIndex] THEN
				BwLimitsEnabled:=FALSE;
			END_IF
		END_IF
	END_FOR
END_FOR

AxisController.bFwEnabled:=FwLimitsEnabled;		//Feedback to ST_AxisControl that forward positioning is available
AxisController.bBwEnabled:=BwLimitsEnabled;		//Feedback to ST_AxisControl that backward positioning is available

//////////////////////////////////////////////////////////
//  ____   _____        _______ ____    _   _ ____  	//
// |  _ \ / _ \ \      / | ____|  _ \  | | | |  _ \ 	//
// | |_) | | | \ \ /\ / /|  _| | |_) | | | | | |_) |	//
// |  __/| |_| |\ V  V / | |___|  _ <  | |_| |  __/ 	//
// |_|    \___/  \_/\_/  |_____|_| \_\  \___/|_|   		//
//														//
/////////////////////////////////////////////////////////// 
(*
Power up the axis.
Externally fed variables are bEnabled and fOverride, limits all controlled internally.
*)                                           
MCPower(
	Axis:=AxisController.Axis,
	Enable:=AxisController.bEnable,
	Enable_Positive:=FwLimitsEnabled,
	Enable_Negative:=BwLimitsEnabled,
	Override:=AxisController.fOverride,
	Status=>,
	Busy=>, 
	Active=>AxisController.bAxisReady,	//Maybe want a bPowered or bEnabled flag instead?
	Error=>,
	ErrorID=>
);

//////////////////////////////////////////////////////////////////////////////////////////////////////////
//  ____  _____    _    ____    ____   _    ____     _    __  __ _____ _____ _____ ____  ____  			//
// |  _ \| ____|  / \  |  _ \  |  _ \ / \  |  _ \   / \  |  \/  | ____|_   _| ____|  _ \/ ___| 			//
// | |_) |  _|   / _ \ | | | | | |_) / _ \ | |_) | / _ \ | |\/| |  _|   | | |  _| | |_) \___ \ 			//
// |  _ <| |___ / ___ \| |_| | |  __/ ___ \|  _ < / ___ \| |  | | |___  | | | |___|  _ < ___) |			//
// |_| \_|_____/_/   \_|____/  |_| /_/   \_|_| \_/_/   \_|_|  |_|_____| |_| |_____|_| \_|____/ 			//
//                                                                                           			//
//////////////////////////////////////////////////////////////////////////////////////////////////////////
(*
Check NC parameters available from MCReadParameter FB (17 in total)
See eRWParameter DUT for complete list or PLC OPEN documentation
To call all 17 from a single functionblock instance only 1 can be checked per cycle so there will be at minimum a 34 cycle delay checking each parameter
The MCReadParameter does also cover the functionality of MCReadBoolParameter so these booleans are separately converted from the MCReadParameter call
*)
MCReadParameter(Axis:=AxisController.AXIS,ParameterNumber:=iParam);
IF MCReadParameter.Valid THEN
	MCReadParameter.Enable:=FALSE;
	AxisController.fParameters[iParam]:=MCReadParameter.Value;
	iParam:= iParam+1;
	IF iParam>17 THEN
		iParam:=1;
	END_IF
ELSE
	MCReadParameter.Enable:=TRUE;
END_IF

//Convert LREALS to BOOLS


IF AxisController.fParameters[eRWParameter.EnableLimitPos]=1 THEN
	AxisController.bSoftLimPosEn:=TRUE;
ELSE
	AxisController.bSoftLimPosEn:=FALSE;
END_IF
IF AxisController.fParameters[eRWParameter.EnableLimitNeg]=1 THEN
	AxisController.bSoftLimNegEn:=TRUE;
ELSE
	AxisController.bSoftLimNegEn:=FALSE;
END_IF
IF AxisController.fParameters[eRWParameter.EnablePosLagMonitoring]=1 THEN
	AxisController.bPosLagEn:=TRUE;
ELSE
	AxisController.bPosLagEn:=FALSE;
END_IF

//////////////////////////////////////////////////////////////////////////////////////////////////////////
//  __  __  ____   _____ _   _ _   _  ____ _____ ___ ___  _   _    ____    _    _     _     ____  		//
// |  \/  |/ ___| |  ___| | | | \ | |/ ___|_   _|_ _/ _ \| \ | |  / ___|  / \  | |   | |   / ___| 		//
// | |\/| | |     | |_  | | | |  \| | |     | |  | | | | |  \| | | |     / _ \ | |   | |   \___ \ 		//
// | |  | | |___  |  _| | |_| | |\  | |___  | |  | | |_| | |\  | | |___ / ___ \| |___| |___ ___) |		//
// |_|  |_|\____| |_|    \___/|_| \_|\____| |_| |___\___/|_| \_|  \____/_/   \_|_____|_____|____/ 		//
//                                         																//                                                      
//////////////////////////////////////////////////////////////////////////////////////////////////////////
(*
Call MC Function Blocks and clear execute signals
Any MC function blocks added to the state machine must be called here with the given format.
Some FBs have slightly differing structures so these should aim to conform to the existing structure
Function blocks will hold done and error signals for 1 cycle with no execute held
*)
MCReadParameter(Axis:=AxisController.Axis);	//Reading in motion parameters, using one functionblock for all params means need to disable

MCReset(Axis:=AxisController.Axis);
MCReset.Execute:=FALSE;

MCWriteParameter(Axis:=AxisController.Axis);
MCWriteParameter.Execute:=FALSE;

MCWriteBoolParameter(Axis:=AxisController.Axis);
MCWriteBoolParameter.Execute:=FALSE;

MCSetPosition(Axis:=AxisController.Axis);
MCSetPosition.Execute:=FALSE;

MCMoveAbsolute(Axis:=AxisController.Axis);
MCMoveAbsolute.Execute:=FALSE;

MCMoveRelative(Axis:=AxisController.Axis);
MCMoveRelative.Execute:=FALSE;

MCGearIn(Slave:=AxisController.Axis, Master:=GVL.axes[AxisController.masterAxis].Axis);
MCGearIn.Execute:=FALSE;

MCGearInMultiMaster(Master1:=GVL.axes[AxisController.masterAxes[1].i].Axis,Master2:=GVL.axes[AxisController.masterAxes[2].i].Axis,Master3:=GVL.axes[AxisController.masterAxes[3].i].Axis,Master4:=GVL.axes[AxisController.masterAxes[4].i].Axis,Slave:=AxisController.Axis);
MCGearInMultiMaster.Enable:=FALSE;	//NOT EXECUTE AS FB ALLOWS CONTINUAL UPDATING OF RATIOS WHILST ENABLED

MCGearOut(Slave:=AxisController.Axis);
MCGearOut.Execute:=FALSE;

MCJog(Axis:=AxisController.Axis);
MCJog.JogBackwards:=FALSE;
MCJog.JogForward:=FALSE;

MCStepAbsoluteSwitch(Axis:=AxisController.Axis,Parameter:=MCHomingParameter);
MCStepAbsoluteSwitch.Execute:=FALSE;

MCFinishHoming(Axis:=AxisController.Axis,Parameter:=MCHomingParameter);
MCFinishHoming.Execute:=FALSE;

MCMoveVelocity(Axis:=AxisController.Axis);
MCMoveVelocity.Execute:=FALSE;

MCStop(Axis:=AxisController.Axis);
MCStop.Execute:=FALSE;

//////////////////////////////////////////////////////////////////////////////////////////////////////////////////////////////////////////////
//   ____ ___  __  __ __  __    _    _   _ ____     ____    _    ____  _____   ____ _____  _  _____ _____ __  __ _____ _   _ _____ ____ 	// 
//  / ___/ _ \|  \/  |  \/  |  / \  | \ | |  _ \   / ___|  / \  / ___|| ____| / ___|_   _|/ \|_   _| ____|  \/  | ____| \ | |_   _/ ___| 	//
// | |  | | | | |\/| | |\/| | / _ \ |  \| | | | | | |     / _ \ \___ \|  _|   \___ \ | | / _ \ | | |  _| | |\/| |  _| |  \| | | | \___ \ 	//
// | |__| |_| | |  | | |  | |/ ___ \| |\  | |_| | | |___ / ___ \ ___) | |___   ___) || |/ ___ \| | | |___| |  | | |___| |\  | | |  ___) |	//
//  \____\___/|_|  |_|_|  |_/_/   \_|_| \_|____/   \____/_/   \_|____/|_____| |____/ |_/_/   \_|_| |_____|_|  |_|_____|_| \_| |_| |____/	//
//																																			//
//////////////////////////////////////////////////////////////////////////////////////////////////////////////////////////////////////////////

(*
Internal statemachine to handle motion control flow and logic.
Functions are NOT called in this statemachine, these just update values given to the state machine. This was the method recommended by Beckhoff
The following basic wrapper should be used for adding new function blocks. Any that do not conform to this should be modified to conform
Notably some FBs have no .Done but do have .Active
	
	mcFunctionBlock.Execute		:=AxisController.bExecute;
	mcFunctionBlock.misc1..n	:=AxisController.misc1..n;
	
	bDone:=mcFunctionBlock.Done;
	AxisController.bBusy:= mcFunctionBlock.Busy;
	
	If mcFunctionBlock.Error THEN
		AxisController.bError:=TRUE;
		AxisController.iErrorID:= mcFunctionBlock.ErrorID;
	END_IF
	IF NOT mcFunctionBlock.Busy THEN
		eCommandLatched:=eMcCommand.Idle;
	END_IF
	
Function block specific parameters should be added to the ST_AxisControl if not already listed
eCommandLatched is currently being used to hold control flow logic so that users cannot send new commands until previous ones have complete.
This will definitely need to be modified to allow buffering in the future and to allow stop/halt commands 
but I haven't looked in to the best way to do this yet.	

It may be that it doesn't matter if it is latched at all as we can rely on waiting for the done signal before sending subsequent commands if it really matters
*)
//If we're not doing anything or have just done something we no longer latch on the given command
IF NOT AxisController.AXIS.Status.HasJob OR AxisController.bDone THEN
	eCommandLatched:=AxisController.eCommand;
END_IF
CASE eCommandLatched OF
	
	eMcCommand.Idle:
		AxisController.bBusy	:=FALSE;
		AxisController.bExecute	:=FALSE;
///////////////////////////////////////////////////////////////////////////////////////////////////////////////////////////////	
	eMcCommand.Reset:
		AxisController.bError	:=FALSE;
		MCReset.Execute:=AxisController.bReset;
		
		bDone:=McReset.Done;
		AxisController.bBusy:=MCReset.Busy;
		IF MCReset.Error THEN
			AxisController.bError:=TRUE;
			AxisController.iErrorID:=MCReset.ErrorID;	
		END_IF
		IF NOT MCReset.Busy THEN
			eCommandLatched:=eMcCommand.Idle;
			AxisController.bReset:=FALSE;
		END_IF
///////////////////////////////////////////////////////////////////////////////////////////////////////////////////////////////
	eMcCommand.WriteParameter:		
		MCWriteParameter.Execute:=AxisController.bExecute;
		MCWriteParameter.ParameterNumber:=AxisController.iParameterIndex;
		MCWriteParameter.Value:=AxisController.fParameterValue;
		
		bDone:=MCWriteParameter.Done;
		AxisController.bBusy:= MCWriteParameter.Busy;
		
		IF MCWriteParameter.Error THEN
			AxisController.bError:=TRUE;
			AxisController.iErrorID:=MCWriteParameter.ErrorID;	
		END_IF	
		IF NOT MCWriteParameter.Busy THEN
			eCommandLatched:=eMcCommand.Idle;
		END_IF			
///////////////////////////////////////////////////////////////////////////////////////////////////////////////////////////////
	eMcCommand.WriteBoolParameter:	
		MCWriteBoolParameter.Execute:=AxisController.bExecute;
		MCWriteBoolParameter.ParameterNumber:=AxisController.iParameterIndex;
		MCWriteBoolParameter.Value:=AxisController.bInput;
		
		bDone:=MCWriteBoolParameter.Done;
		AxisController.bBusy:=MCWriteBoolParameter.Busy;
		
		IF MCWriteBoolParameter.Error THEN
			AxisController.bError:= TRUE;
			AxisController.iErrorID:=MCWriteBoolParameter.ErrorID;
		END_IF			
		IF NOT MCWriteBoolParameter.Busy THEN
			eCommandLatched:=eMcCommand.Idle;
		END_IF	
///////////////////////////////////////////////////////////////////////////////////////////////////////////////////////////////
	eMcCommand.SetPosition:	
		MCSetPosition.Execute:=AxisController.bExecute;
		MCSetPosition.Position:=AxisController.fPosition;
		
		AxisController.bBusy:=MCSetPosition.Busy;
		bDone:=MCSetPosition.Done;
		
		IF MCSetPosition.Error THEN
			AxisController.bError:=TRUE;
			AxisController.iErrorID:= MCSetPosition.ErrorID;
		END_IF
		IF NOT MCSetPosition.Busy THEN
			eCommandLatched:=eMcCommand.Idle;
		END_IF
///////////////////////////////////////////////////////////////////////////////////////////////////////////////////////////////
	eMcCommand.MoveAbsolute:	
		MCMoveAbsolute.Execute:=AxisController.bExecute;
		MCMoveAbsolute.Position:=AxisController.fPosition;
		MCMoveAbsolute.Velocity:=AxisController.fVelocity;
		MCMoveAbsolute.Acceleration:=AxisController.fAcceleration;
		MCMoveAbsolute.Deceleration:=AxisController.fDeceleration;
		MCMoveAbsolute.Jerk:=0;
		MCMoveAbsolute.BufferMode:=MC_BufferMode.MC_Buffered;
		
		bDone:=MCMoveAbsolute.Done;
		AxisController.bBusy:=MCMoveAbsolute.Busy;
		
		IF MCMoveAbsolute.Error THEN
			AxisController.bError:=TRUE;
			AxisController.iErrorID:=MCMoveAbsolute.ErrorID;
		END_IF
		IF NOT MCMoveAbsolute.Busy THEN
			eCommandLatched:=eMcCommand.Idle;
		END_IF
///////////////////////////////////////////////////////////////////////////////////////////////////////////////////////////////
	eMcCommand.MoveRelative:		
		MCMoveRelative.Execute:=AxisController.bExecute;
		MCMoveRelative.Distance:=AxisController.fDistance;
		MCMoveRelative.Velocity:=AxisController.fVelocity;
		MCMoveRelative.Acceleration:=AxisController.fAcceleration;
		MCMoveRelative.Deceleration:=AxisController.fDeceleration;
		MCMoveRelative.Jerk:=0;
		MCMoveRelative.BufferMode:=MC_BufferMode.MC_Buffered;
		
		bDone:=MCMoveRelative.Done;
		AxisController.bBusy:=MCMoveRelative.Busy;
		
		IF MCMoveRelative.Error THEN
			AxisController.bError:=TRUE;
			AxisController.iErrorID:=MCMoveRelative.ErrorID;
		END_IF
		IF NOT MCMoveRelative.Busy THEN
			eCommandLatched:=eMcCommand.Idle;
		END_IF		
///////////////////////////////////////////////////////////////////////////////////////////////////////////////////////////////
	eMcCommand.GearIn:
		//Dependent on +ve or -ve gear ratio determines whether to link Fw to Fw and Bw to Bw or Fw to Bw and Bw to Fw
		IF AxisController.fGearRatioNum>0 THEN
			Limits.coupledFwLimit[GVL.iAxis][1].eLimitType:=eLimitCoupling.FwSw;		
			Limits.coupledBwLimit[GVL.iAxis][1].eLimitType:=eLimitCoupling.BwSw;				
		END_IF
		IF AxisController.fGearRatioNum<0 THEN
			Limits.coupledFwLimit[GVL.iAxis][1].eLimitType:=eLimitCoupling.BwSw;
			Limits.coupledBwLimit[GVL.iAxis][1].eLimitType:=eLimitCoupling.FwSw;		
		END_IF
		Limits.coupledFwLimit[GVL.iAxis][1].iMasterAxis:=AxisController.masterAxis;
		Limits.coupledBwLimit[GVL.iAxis][1].iMasterAxis:=AxisController.masterAxis;
		
		MCGearIn.Execute:=AxisController.bExecute;
		MCGearIn.RatioNumerator:=AxisController.fGearRatioNum;
		MCGearIn.RatioDenominator:=AxisController.iGearRatioDen;
		
		bDone:=McGearIn.InGear;
		AxisController.bBusy:=MCGearIn.Busy;
		
		IF MCGearIn.Error THEN
			AxisController.bError:=TRUE;
			AxisController.iErrorID:=MCGearIn.ErrorID;
		END_IF		
		IF NOT MCGearIn.Busy THEN
			eCommandLatched:=eMcCommand.Idle;
		END_IF
///////////////////////////////////////////////////////////////////////////////////////////////////////////////////////////////
	eMcCommand.GearInMultiMaster:		
		//Set up limits
		FOR iMasterIndex:=1 TO GVL.axisCoupleMax DO
			IF AxisController.masterAxes[iMasterIndex].ratio>0 THEN
				Limits.coupledFwLimit[GVL.iAxis][iMasterIndex+1].eLimitType:=eLimitCoupling.FwSw;				
				Limits.coupledBwLimit[GVL.iAxis][iMasterIndex+1].eLimitType:=eLimitCoupling.BwSw;				
			END_IF
			IF AxisController.masterAxes[iMasterIndex].ratio<0 THEN
				Limits.coupledFwLimit[GVL.iAxis][iMasterIndex+1].eLimitType:=eLimitCoupling.BwSw;
				Limits.coupledBwLimit[GVL.iAxis][iMasterIndex+1].eLimitType:=eLimitCoupling.FwSw;
			END_IF
			Limits.coupledFwLimit[GVL.iAxis][iMasterIndex+1].iMasterAxis:=AxisController.masterAxes[iMasterIndex].i;
			Limits.coupledBwLimit[GVL.iAxis][iMasterIndex+1].iMasterAxis:=AxisController.masterAxes[iMasterIndex].i;
		END_FOR
		

		
		(*	Issue with this MC block (other than everything...) is that it doesn't conform to the standard and use an execute signal. The execute
			signal in any other block determines that when it is high one of either error,done,busy must be on. That is not the case with this block
			what happens is it triggers, doesn't register a busy and so immediately clears as done. If has been modified to conform.
		*)
		MCGearInMultiMaster.Enable:=AxisController.bExecute;
		MCGearInMultiMaster.GearRatio1:=AxisController.masterAxes[1].ratio;
		MCGearInMultiMaster.GearRatio2:=AxisController.masterAxes[2].ratio;
		MCGearInMultiMaster.GearRatio3:=AxisController.masterAxes[3].ratio;
		MCGearInMultiMaster.GearRatio4:=AxisController.masterAxes[4].ratio;
		
		AxisController.bBusy:=MCGearInMultiMaster.Busy;
		IF MCGearInMultiMaster.Enable THEN
			AxisController.bBusy:=TRUE;	//busy does not go immediately high when enable high 
			bDone:=FALSE;
		END_IF

		bDone:=MCGearInMultiMaster.InGear;	
		IF MCGearInMultiMaster.Error THEN
			AxisController.bError:=TRUE;
			AxisController.iErrorID:=MCGearInMultiMaster.ErrorID;
		END_IF
		IF NOT MCGearInMultiMaster.Busy THEN
			eCommandLatched:=eMcCommand.Idle;
		END_IF
///////////////////////////////////////////////////////////////////////////////////////////////////////////////////////////////
	eMcCommand.GearOut:		
		//Gearout - remove all masters from slave
		FOR iMasterIndex:=1 TO 5 DO
				Limits.coupledFwLimit[GVL.iAxis][iMasterIndex].eLimitType:=eLimitCoupling.None;
				Limits.coupledBwLimit[GVL.iAxis][iMasterIndex].eLimitType:=eLimitCoupling.None;
		END_FOR		
	
		MCGearOut.Execute:=AxisController.bExecute;
		
		AxisController.bBusy:=MCGearOut.Busy;
		bDone:=MCGearOut.Done;
		IF MCGearOut.Error THEN
			AxisController.bError:=TRUE;
			AxisController.iErrorID:=MCGearOut.ErrorID;
		END_IF
		IF NOT MCGearOut.Busy THEN
			eCommandLatched:=eMcCommand.Idle;
		END_IF
	///////////////////////////////////////////////////////////////////////////////////////////////////////////////////////////////			
	eMcCommand.Jog:
		MCJog.JogForward:=AxisController.bJogForward;
		MCJog.JogBackwards:=AxisController.bJogBackward;
		
		bDone:=MCJog.Done;
		
		IF MCJog.Error THEN
			AxisController.bError:=TRUE;
			AxisController.iErrorID:=MCJog.ErrorID;
		END_IF
		IF NOT MCJog.Busy THEN
			eCommandLatched:=eMcCommand.Idle;
		END_IF
	///////////////////////////////////////////////////////////////////////////////////////////////////////////////////////////////	
	eMcCommand.HomeStepAbsoluteSwitch:
		//Issue: If execute not held high the function will not reverse on its own to find the abs switch when hitting a limit
		//You have to reissue the command. I want to try and keep bExecute high
		IF (NOT Limits.FwLimit[GVL.iAxis]) OR (NOT Limits.BwLimit[GVL.iAxis]) THEN
			MCStepAbsoluteSwitch.Execute:=TRUE;
		ELSE	
			MCStepAbsoluteSwitch.Execute:=AxisController.bExecute;
		END_IF
	
		MCStepAbsoluteSwitch.Direction:= AxisController.mcHomeDirection;
		MCStepAbsoluteSwitch.SwitchMode:=AxisController.mcSwitchMode;
		MCStepAbsoluteSwitch.ReferenceSignal:=AxisController.mcSignalRef;
		MCStepAbsoluteSwitch.Velocity:=AxisController.fHomeVelocity;
		MCStepAbsoluteSwitch.Acceleration:=0;
		MCStepAbsoluteSwitch.Deceleration:=0;
		MCStepAbsoluteSwitch.Jerk:=0;
		MCStepAbsoluteSwitch.TorqueLimit:=AxisController.fHomeTorque;
		MCStepAbsoluteSwitch.SetPosition:=AxisController.fHomePosition;
		MCStepAbsoluteSwitch.TimeLimit:=AxisController.tHomeTimeLimit;
		MCStepAbsoluteSwitch.DistanceLimit:=AxisController.fHomeDistanceLimit;
		MCStepAbsoluteSwitch.PositiveLimitSwitch:= NOT Limits.FwLimit[GVL.iAxis];	//Step FB has R_TRIG behaviour but limits set as Normally Closed so logic is inverted
		MCStepAbsoluteSwitch.NegativeLimitSwitch:= NOT Limits.BwLimit[GVL.iAxis];	//Step FB has R_TRIG behaviour but limits set as Normally Closed so logic is inverted
		MCStepAbsoluteSwitch.BufferMode:=AxisController.buffer;
		StOptions4.DisableDriveAccess:=TRUE;		//Testing required with hardware. This step may be redundant.
		MCStepAbsoluteSwitch.Options:=StOptions4;
		
		bDone:=MCStepAbsoluteSwitch.Done;
		AxisController.bBusy:=MCStepAbsoluteSwitch.Busy;
		
		IF MCStepAbsoluteSwitch.Error THEN
			AxisController.bError:=TRUE;
			AxisController.iErrorID:=MCStepAbsoluteSwitch.ErrorID;
		END_IF
		IF NOT MCStepAbsoluteSwitch.Busy THEN
			eCommandLatched:=eMcCommand.Idle;
		END_IF
	///////////////////////////////////////////////////////////////////////////////////////////////////////////////////////////////	
	eMcCommand.HomeFinish:
		MCFinishHoming.Execute:=AxisController.bExecute;
		MCFinishHoming.Distance:=AxisController.fHomeDistance;
		MCFinishHoming.Velocity:=AxisController.fHomeVelocity;
		
		StOptions2.DisableDriveAccess:=TRUE;	//Testing required with hardware. This step may be redundant.
		MCFinishHoming.Options:=StOptions2;
		
		bDone:=MCFinishHoming.Done;
		AxisController.bBusy:=MCFinishHoming.Busy;
		
		IF MCFinishHoming.Error THEN
			AxisController.bError:=TRUE;
			AxisController.iErrorID:=MCFinishHoming.ErrorID;
		END_IF
		IF NOT MCFinishHoming.Busy THEN
			eCommandLAtched:=eMcCommand.Idle;
		END_IF
	///////////////////////////////////////////////////////////////////////////////////////////////////////////////////////////////	
	eMcCommand.MoveVelocity:
		MCMoveVelocity.Execute:=AxisController.bExecute;
		MCMoveVelocity.Acceleration:=AxisController.fAcceleration;
		MCMoveVelocity.Deceleration:=AxisController.fDeceleration;
		
		//Simple logic to allow negative velocity inputs rather than having to set the direction object
		IF AxisController.fVelocity>= 0 THEN
			MCMoveVelocity.Velocity:=AxisController.fVelocity;
			MCMoveVelocity.Direction:= MC_Positive_Direction;
		ELSE
			MCMoveVelocity.Velocity:=ABS(AxisController.fVelocity);
			MCMoveVelocity.Direction:= MC_Negative_Direction;
		END_IF
		
		bDone:=MCMoveVelocity.InVelocity;
		AxisController.bBusy:=MCMoveVelocity.Busy;
		
		IF MCMoveVelocity.Error THEN
			AxisController.bError:=TRUE;
			AxisController.iErrorID:=MCMoveVelocity.ErrorID;
		END_IF
		IF NOT MCMoveVelocity.Busy THEN
			eCommandLatched:=eMcCommand.Idle;
		END_IF
	///////////////////////////////////////////////////////////////////////////////////////////////////////////////////////////////	
	eMcCommand.Stop:
		McStop.Execute:=AxisController.bExecute;
		McStop.Deceleration:=AxisController.fDeceleration;
		McStop.Jerk:=0;
		
		bDone:=McStop.Done;
		AxisController.bBusy:=McStop.Busy;
		
		IF MCStop.Error THEN
			AxisController.bError:= TRUE;
			AxisController.iErrorID:=MCStop.ErrorId;
		END_IF
		IF	NOT MCStop.Busy THEN
			eCommandLatched:=eMcCommand.Idle;
		END_IF
		
END_CASE

////////////////////////////////////////// 
//  _____ _        _    ____ ____  		//
// |  ___| |      / \  / ___/ ___| 		//
// | |_  | |     / _ \| |  _\___ \ 		//
// |  _| | |___ / ___ | |_| |___) |		//
// |_|   |_____/_/   \_\____|____/ 		//
//                                		//
//////////////////////////////////////////
AxisController.bMoving:=AxisController.Axis.Status.Moving;	
AxisController.bExecute:=FALSE;

(*
As we never hold Execute high, the done signal from each function block will only stay on for 1 cycle tick
The following logic just uses an SR latch to hold this done signal TRUE until it is cleared either by an error or the axis going busy

Errors are always latched as they are only ever set by a FB error and cleared by a reset command
*)
doneLatch(SET1:=bDone,RESET:=(AxisController.bBusy OR AxisController.bError));
AxisController.bDone:=doneLatch.Q1;

END_FUNCTION_BLOCK

// ---- GlobalTextList.TcGTLO
TEXTLIST GlobalTextList
  100 = ' ADVANCED HOMING '
  94 = ' DISCRETE MOVES '
  91 = ' GEARING '
  92 = ' MULTI-GEARING '
  90 = ' PARAMETERS '
  126 = ' Parameters '
  124 = ' POWER '
  115 = ' Simulation '
  17 = '%2.2f'
  37 = '%3.2f'
  16 = '%4.2f'
  11 = '%5.2f'
  12 = '%5.4f'
  31 = '%d'
  0 = '%f'
  15 = '%f4.2'
  2 = '%f5.2'
  69 = '%s'
  79 = '+'
  80 = '-'
  82 = ':'
  25 = 'ABS.MOVE'
  118 = 'Absolute Flag High Position'
  119 = 'Absolute Flag Low Position'
  5 = 'Absolute Position'
  6 = 'ABSOLUTE POSITION:'
  53 = 'ActualVelocity'
  106 = 'Adv. Homing'
  20 = 'AXIS %d'
  19 = 'AXIS %f'
  29 = 'AXIS BUSY'
  121 = 'AXIS NAME:'
  21 = 'AXIS SELECT'
  22 = 'AXIS SELECT:'
  120 = 'AXIS SELECTION:'
  14 = 'BW'
  123 = 'BW ENABLED'
  111 = 'CALIBRATED'
  87 = 'Casd'
  3 = 'CMD 28'
  40 = 'CMD POSITION:'
  44 = 'Cmd Position:'
  54 = 'CommandedVelocity'
  4 = 'CommandList.28'
  99 = 'Continuous\nMotion'
  27 = 'COUPLED'
  33 = 'DEN.'
  107 = 'Disable MC'
  39 = 'DISCRETE MOVES'
  10 = 'DISTANCE'
  7 = 'DISTANCE:'
  103 = 'Distance:'
  63 = 'DONE'
  18 = 'EN'
  49 = 'En/Dis'
  71 = 'ENABLE H'
  70 = 'ENABLE V'
  62 = 'ERROR'
  105 = 'FINISH HOMING'
  13 = 'FW'
  122 = 'FW ENABLED'
  34 = 'GEAR IN'
  36 = 'GEAR OUT'
  35 = 'GEARED'
  38 = 'GEARING'
  93 = 'Gearing'
  1 = 'GO'
  86 = 'HC:'
  85 = 'HG:'
  116 = 'High Limit Position'
  76 = 'HORIZONTAL CENTRE'
  75 = 'HORIZONTAL GAP'
  95 = 'I/O'
  78 = 'Jog Backwards'
  77 = 'Jog Forwards'
  117 = 'Low Limit Position'
  65 = 'MASTER1:'
  66 = 'MASTER2:'
  67 = 'MASTER3:'
  125 = 'MASTER4:'
  30 = 'MASTER:'
  56 = 'MaxAccelerationAppl'
  55 = 'MaxAccelerationSystem'
  59 = 'MaxDecelerationAppl'
  58 = 'MaxDecelerationSystem'
  61 = 'MaxJerkAppl'
  60 = 'MaxJerkSystem'
  47 = 'MaxPositionLag'
  50 = 'MaxVelocity System'
  57 = 'MaxVelocityAppl'
  52 = 'MaxVelocityApplication'
  51 = 'MaxVelocitySystem'
  28 = 'MOVING'
  64 = 'MULTI-GEARING'
  32 = 'NUM.'
  41 = 'Parameters'
  42 = 'PARAMETERS'
  9 = 'POWER'
  68 = 'RATIO:'
  24 = 'RB POSITION:'
  885 = 'Read Position:'
  26 = 'REL.MOVE'
  8 = 'RESET'
  48 = 'SET'
  102 = 'Set Position:'
  108 = 'Simulate Abs'
  112 = 'Simulate AbsSw/Pulse'
  110 = 'Simulate NegLim'
  109 = 'Simulate PosLim'
  113 = 'Simulated Axis'
  114 = 'Simulation'
  88 = 'Single Axis'
  89 = 'Slit Set'
  104 = 'STEP ABS SW'
  1060 = 'STEP LIMIT SW'
  598 = 'STEP REF. PULSE (NO EDGE DETECTION)'
  229 = 'STOP'
  46 = 'SWLimitNeg:'
  43 = 'SWLimitPos'
  45 = 'SWLimitPos:'
  98 = 'Synchronised\nMotion'
  96 = 'Synchronised Motion'
  97 = 'SynchronisedMotion'
  72 = 'Toggle'
  84 = 'VC:'
  973 = 'VELOCITY'
  1158 = 'Velocity'
  662 = 'VELOCITY MOVE'
  23 = 'VELOCITY:'
  101 = 'Velocity:'
  74 = 'VERTICAL CENTRE'
  73 = 'VERTICAL GAP'
  81 = 'VG'
  83 = 'VG:'
END_TEXTLIST

// ---- VISUs/COMMAND VISUS/Gearing.TcVIS
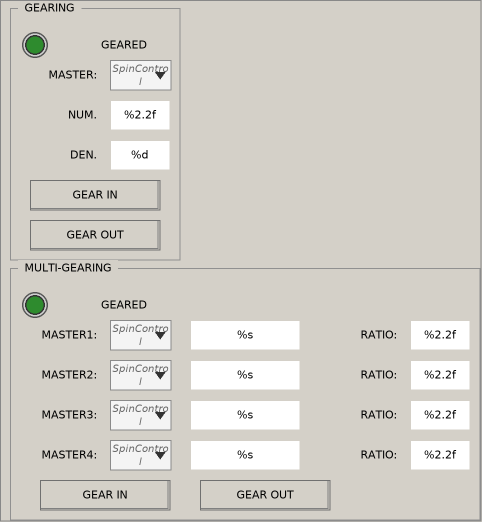
VISUALIZATION Gearing  // 482x522
    GroupBox (10,0 170x260), "GEARING"
        Textfield (40,30 100x30), "GEARED", text variable: MAIN.hmiAxisSelect
        SpinControl (100,60 61x30), variable: GVL.axes[MAIN.hmiAxisSelect].masterAxis
            p651134158: GVL.axisNumMax
            OnMouseClick: write GVL.axes[MAIN.hmiAxisSelect].masterAxis via Default
        Textfield (10,60 80x30), "MASTER:", text variable: MAIN.hmiAxisSelect
        Textfield (100,100 60x30), "%2.2f", text variable: GVL.axes[MAIN.hmiAxisSelect].fGearRatioNum
            OnMouseClick: write GVL.axes[MAIN.hmiAxisSelect].fGearRatioNum via Default
        Textfield (10,100 80x30), "NUM.", text variable: MAIN.hmiAxisSelect
        Textfield (100,140 60x30), "%d", text variable: GVL.axes[MAIN.hmiAxisSelect].iGearRatioDen
            OnMouseClick: write GVL.axes[MAIN.hmiAxisSelect].iGearRatioDen via Default
        Textfield (10,140 80x30), "DEN.", text variable: MAIN.hmiAxisSelect
        Button (20,180 130x30), "GEAR IN"
            OnMouseClick: execute { GVL.axes[MAIN.hmiAxisSelect].eCommand:=eMcCommand.GearIn; GVL.axes[MAIN.hmiAxisSelect].bExecute:= TRUE; }
        Button (20,220 130x30), "GEAR OUT"
            OnMouseClick: execute { GVL.axes[MAIN.hmiAxisSelect].eCommand:=eMcCommand.GearOut; GVL.axes[MAIN.hmiAxisSelect].bExecute:= TRUE; }
        Lamp1 (10,30 30x30), variable: GVL.axes[MAIN.hmiAxisSelect].iAxisState=500, style: Lamp-Lamp1-Green
    GroupBox (10,260 470x260), "MULTI-GEARING"
        Lamp1 (10,30 30x30), variable: GVL.axes[MAIN.hmiAxisSelect].iAxisState=500, style: Lamp-Lamp1-Green
        Textfield (40,30 100x30), "GEARED", text variable: MAIN.hmiAxisSelect
        SpinControl (100,60 61x30), variable: GVL.axes[MAIN.hmiAxisSelect].masterAxes[1].i
            p651134158: GVL.axisNumMax
            OnMouseClick: write GVL.axes[MAIN.hmiAxisSelect].masterAxes[1].i via Default
        Textfield (10,60 80x30), "MASTER1:", text variable: MAIN.hmiAxisSelect
        Textfield (400,60 60x30), "%2.2f", text variable: GVL.axes[MAIN.hmiAxisSelect].masterAxes[1].ratio
            OnMouseClick: write GVL.axes[MAIN.hmiAxisSelect].masterAxes[1].ratio via Default
        Textfield (310,60 80x30), "RATIO:", text variable: MAIN.hmiAxisSelect
        Button (30,220 130x30), "GEAR IN"
            OnMouseClick: execute { GVL.axes[MAIN.hmiAxisSelect].eCommand:=eMcCommand.GearInMultiMaster; GVL.axes[MAIN.hmiAxisSelect].bExecute:= TRUE; }
        Button (190,220 130x30), "GEAR OUT"
            OnMouseClick: execute { GVL.axes[MAIN.hmiAxisSelect].eCommand:=eMcCommand.GearOut; GVL.axes[MAIN.hmiAxisSelect].bExecute:= TRUE; }
        SpinControl (100,100 61x30), variable: GVL.axes[MAIN.hmiAxisSelect].masterAxes[2].i
            p651134158: GVL.axisNumMax
            OnMouseClick: write GVL.axes[MAIN.hmiAxisSelect].masterAxes[2].i via Default
        SpinControl (100,140 61x30), variable: GVL.axes[MAIN.hmiAxisSelect].masterAxes[3].i
            p651134158: GVL.axisNumMax
            OnMouseClick: write GVL.axes[MAIN.hmiAxisSelect].masterAxes[3].i via Default
        SpinControl (100,180 61x30), variable: GVL.axes[MAIN.hmiAxisSelect].masterAxes[4].i
            p651134158: GVL.axisNumMax
            OnMouseClick: write GVL.axes[MAIN.hmiAxisSelect].masterAxes[4].i via Default
        Textfield (310,100 80x30), "RATIO:", text variable: MAIN.hmiAxisSelect
        Textfield (310,140 80x30), "RATIO:", text variable: MAIN.hmiAxisSelect
        Textfield (310,180 80x30), "RATIO:", text variable: MAIN.hmiAxisSelect
        Textfield (10,100 80x30), "MASTER2:", text variable: MAIN.hmiAxisSelect
        Textfield (10,140 80x30), "MASTER3:", text variable: MAIN.hmiAxisSelect
        Textfield (10,180 80x30), "MASTER4:", text variable: MAIN.hmiAxisSelect
        Textfield (400,100 60x30), "%2.2f", text variable: GVL.axes[MAIN.hmiAxisSelect].masterAxes[2].ratio
            OnMouseClick: write GVL.axes[MAIN.hmiAxisSelect].masterAxes[2].ratio via Default
        Textfield (400,140 60x30), "%2.2f", text variable: GVL.axes[MAIN.hmiAxisSelect].masterAxes[3].ratio
            OnMouseClick: write GVL.axes[MAIN.hmiAxisSelect].masterAxes[3].ratio via Default
        Textfield (400,180 60x30), "%2.2f", text variable: GVL.axes[MAIN.hmiAxisSelect].masterAxes[4].ratio
            OnMouseClick: write GVL.axes[MAIN.hmiAxisSelect].masterAxes[4].ratio via Default
        Textfield (180,60 110x30), "%s", text variable: GVL.axes[GVL.axes[MAIN.hmiAxisSelect].masterAxes[1].i].sAxisName
        Textfield (180,100 110x30), "%s", text variable: GVL.axes[GVL.axes[MAIN.hmiAxisSelect].masterAxes[2].i].sAxisName
        Textfield (180,140 110x30), "%s", text variable: GVL.axes[GVL.axes[MAIN.hmiAxisSelect].masterAxes[3].i].sAxisName
        Textfield (180,180 110x30), "%s", text variable: GVL.axes[GVL.axes[MAIN.hmiAxisSelect].masterAxes[4].i].sAxisName
END_VISUALIZATION

// ---- VISUs/COMMAND VISUS/Parameters.TcVIS
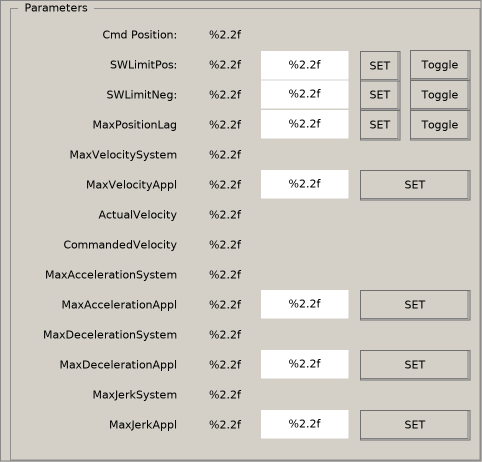
VISUALIZATION Parameters  // 482x462
    GroupBox (10,0 470x460), "Parameters"
        Textfield (170,20 90x30), "%2.2f", text variable: GVL.axes[MAIN.hmiAxisSelect].fParameters[1]
        Textfield (10,50 160x30), "SWLimitPos:"
        Textfield (10,20 160x30), "Cmd Position:"
        Textfield (170,50 90x30), "%2.2f", text variable: GVL.axes[MAIN.hmiAxisSelect].fParameters[2], input disabled if: NOT GVL.axes[MAIN.hmiAxisSelect].bSoftLimPosEn
        Textfield (170,80 90x30), "%2.2f", text variable: GVL.axes[MAIN.hmiAxisSelect].fParameters[3], input disabled if: NOT GVL.axes[MAIN.hmiAxisSelect].bSoftLimNegEn
        Textfield (250,79 89x30), "%2.2f", text variable: GVL.SwLimitNeg
            OnMouseClick: write GVL.SwLimitNeg via Default
        Button (350,80 40x30), "SET"
            toggle GVL.axes[MAIN.hmiAxisSelect].bEXECUTE
            OnMouseClick: execute {
                GVL.axes[Main.hmiAxisSelect].eCommand:=eMcCommand.WriteParameter;
                GVL.axes[Main.hmiAxisSelect].fParameterValue:=GVL.SwLimitNeg;
                GVL.axes[Main.hmiAxisSelect].iParameterIndex:=eRWParameter.SWLimitNeg;
                GVL.axes[Main.hmiAxisSelect].bExecute:=TRUE;
            }
        Button (400,50 60x30), "Toggle", pressed state: GVL.axes[MAIN.hmiAxisSelect].bSoftLimPosEn, text list: 'ButtonStates', text index: GVL.axes[MAIN.hmiAxisSelect].bSoftLimPosEn
            toggle GVL.axes[MAIN.hmiAxisSelect].bEXECUTE
            OnMouseClick: execute {
                GVL.axes[MAIN.hmiAxisSelect].bInput:=NOT GVL.axes[MAIN.hmiAxisSelect].bSoftLimPosEn;
                GVL.axes[MAIN.hmiAxisSelect].eCommand:=eMcCommand.WriteBoolParameter;
                GVL.axes[MAIN.hmiAxisSelect].iParameterIndex:=eRWParameter.EnableLimitPos;
                GVL.axes[MAIN.hmiAxisSelect].bExecute:=TRUE;
            }
        Button (400,80 60x30), "Toggle", pressed state: GVL.axes[MAIN.hmiAxisSelect].bSoftLimNegEn, text list: 'ButtonStates', text index: GVL.axes[MAIN.hmiAxisSelect].bSoftLimNegEn
            toggle GVL.axes[MAIN.hmiAxisSelect].bEXECUTE
            OnMouseClick: execute {
                GVL.axes[MAIN.hmiAxisSelect].bInput:=NOT GVL.axes[MAIN.hmiAxisSelect].bSoftLimNegEn;
                GVL.axes[MAIN.hmiAxisSelect].eCommand:=eMcCommand.WriteBoolParameter;
                GVL.axes[MAIN.hmiAxisSelect].iParameterIndex:=eRWParameter.EnableLimitNeg;
                GVL.axes[MAIN.hmiAxisSelect].bExecute:=TRUE;
            }
        Textfield (10,110 160x30), "MaxPositionLag"
        Textfield (10,140 160x30), "MaxVelocitySystem"
        Textfield (10,170 160x30), "MaxVelocityAppl"
        Textfield (10,200 160x30), "ActualVelocity"
        Textfield (10,230 160x30), "CommandedVelocity"
        Textfield (170,260 90x30), "%2.2f", text variable: GVL.axes[MAIN.hmiAxisSelect].fParameters[12]
        Textfield (10,290 160x30), "MaxAccelerationAppl"
        Textfield (10,320 160x30), "MaxDecelerationSystem"
        Textfield (10,380 160x30), "MaxJerkSystem"
        Button (350,51 40x30), "SET"
            toggle GVL.axes[MAIN.hmiAxisSelect].bEXECUTE
            OnMouseClick: execute {
                GVL.axes[Main.hmiAxisSelect].eCommand:=eMcCommand.WriteParameter;
                GVL.axes[Main.hmiAxisSelect].fParameterValue:=GVL.SwLimitPos;
                GVL.axes[Main.hmiAxisSelect].iParameterIndex:=eRWParameter.SWLimitPos;
                GVL.axes[Main.hmiAxisSelect].bExecute:=TRUE;
            }
        Textfield (10,80 160x30), "SWLimitNeg:"
        Textfield (170,110 90x30), "%2.2f", text variable: GVL.axes[MAIN.hmiAxisSelect].fParameters[7], input disabled if: NOT GVL.axes[MAIN.hmiAxisSelect].bPosLagEn
        Textfield (250,109 89x30), "%2.2f", text variable: GVL.MaxPositionLag
            OnMouseClick: write GVL.MaxPositionLag via Default
        Button (350,110 40x30), "SET"
            toggle GVL.axes[MAIN.hmiAxisSelect].bEXECUTE
            OnMouseClick: execute {
                GVL.axes[Main.hmiAxisSelect].eCommand:=eMcCommand.WriteParameter;
                GVL.axes[Main.hmiAxisSelect].fParameterValue:=GVL.MaxPositionLag;
                GVL.axes[Main.hmiAxisSelect].iParameterIndex:=eRWParameter.MaxPositionLag;
                GVL.axes[Main.hmiAxisSelect].bExecute:=TRUE;
            }
        Button (400,110 60x30), "Toggle", pressed state: GVL.axes[MAIN.hmiAxisSelect].bPosLagEn, text list: 'ButtonStates', text index: GVL.axes[MAIN.hmiAxisSelect].bPosLagEn
            toggle GVL.axes[MAIN.hmiAxisSelect].bEXECUTE
            OnMouseClick: execute {
                GVL.axes[MAIN.hmiAxisSelect].bInput:=NOT GVL.axes[MAIN.hmiAxisSelect].bPosLagEn;
                GVL.axes[MAIN.hmiAxisSelect].eCommand:=eMcCommand.WriteBoolParameter;
                GVL.axes[MAIN.hmiAxisSelect].iParameterIndex:=eRWParameter.EnablePosLagMonitoring;
                GVL.axes[MAIN.hmiAxisSelect].bExecute:=TRUE;
            }
        Textfield (170,140 90x30), "%2.2f", text variable: GVL.axes[MAIN.hmiAxisSelect].fParameters[8]
        Textfield (170,170 90x30), "%2.2f", text variable: GVL.axes[MAIN.hmiAxisSelect].fParameters[9]
        Textfield (250,169 89x30), "%2.2f", text variable: GVL.MaxVelocityAppl
            OnMouseClick: write GVL.MaxVelocityAppl via Default
        Button (350,170 110x30), "SET"
            toggle GVL.axes[MAIN.hmiAxisSelect].bEXECUTE
            OnMouseClick: execute {
                GVL.axes[Main.hmiAxisSelect].eCommand:=eMcCommand.WriteParameter;
                GVL.axes[Main.hmiAxisSelect].fParameterValue:=GVL.MaxVelocityAppl;
                GVL.axes[Main.hmiAxisSelect].iParameterIndex:=eRWParameter.MaxVelocityAppl;
                GVL.axes[Main.hmiAxisSelect].bExecute:=TRUE;
            }
        Textfield (170,200 90x30), "%2.2f", text variable: GVL.axes[MAIN.hmiAxisSelect].fParameters[10]
        Textfield (170,230 90x30), "%2.2f", text variable: GVL.axes[MAIN.hmiAxisSelect].fParameters[11]
        Textfield (10,260 160x30), "MaxAccelerationSystem"
        Textfield (170,290 90x30), "%2.2f", text variable: GVL.axes[MAIN.hmiAxisSelect].fParameters[13]
        Textfield (250,289 89x30), "%2.2f", text variable: GVL.MaxAccelerationAppl
            OnMouseClick: write GVL.MaxAccelerationAppl via Default
        Button (350,290 110x30), "SET"
            toggle GVL.axes[MAIN.hmiAxisSelect].bEXECUTE
            OnMouseClick: execute {
                GVL.axes[Main.hmiAxisSelect].eCommand:=eMcCommand.WriteParameter;
                GVL.axes[Main.hmiAxisSelect].fParameterValue:=GVL.MaxAccelerationAppl;
                GVL.axes[Main.hmiAxisSelect].iParameterIndex:=eRWParameter.MaxAccelerationAppl;
                GVL.axes[Main.hmiAxisSelect].bExecute:=TRUE;
            }
        Textfield (170,320 90x30), "%2.2f", text variable: GVL.axes[MAIN.hmiAxisSelect].fParameters[14]
        Textfield (10,350 160x30), "MaxDecelerationAppl"
        Textfield (170,350 90x30), "%2.2f", text variable: GVL.axes[MAIN.hmiAxisSelect].fParameters[15]
        Textfield (250,349 89x30), "%2.2f", text variable: GVL.MaxDecelerationAppl
            OnMouseClick: write GVL.MaxDecelerationAppl via Default
        Button (350,350 110x30), "SET"
            toggle GVL.axes[MAIN.hmiAxisSelect].bEXECUTE
            OnMouseClick: execute {
                GVL.axes[Main.hmiAxisSelect].eCommand:=eMcCommand.WriteParameter;
                GVL.axes[Main.hmiAxisSelect].fParameterValue:=GVL.MaxDecelerationAppl;
                GVL.axes[Main.hmiAxisSelect].iParameterIndex:=eRWParameter.MaxDecelerationAppl;
                GVL.axes[Main.hmiAxisSelect].bExecute:=TRUE;
            }
        Textfield (170,380 90x30), "%2.2f", text variable: GVL.axes[MAIN.hmiAxisSelect].fParameters[16]
        Textfield (10,410 160x30), "MaxJerkAppl"
        Textfield (170,410 90x30), "%2.2f", text variable: GVL.axes[MAIN.hmiAxisSelect].fParameters[17]
        Textfield (250,409 89x30), "%2.2f", text variable: GVL.MaxJerkAppl
            OnMouseClick: write GVL.MaxJerkAppl via Default
        Button (350,410 110x30), "SET"
            toggle GVL.axes[MAIN.hmiAxisSelect].bEXECUTE
            OnMouseClick: execute {
                GVL.axes[Main.hmiAxisSelect].eCommand:=eMcCommand.WriteParameter;
                GVL.axes[Main.hmiAxisSelect].fParameterValue:=GVL.MaxJerkAppl;
                GVL.axes[Main.hmiAxisSelect].iParameterIndex:=eRWParameter.MaxJerkAppl;
                GVL.axes[Main.hmiAxisSelect].bExecute:=TRUE;
            }
        Textfield (250,50 89x30), "%2.2f", text variable: GVL.SwLimitPos
            OnMouseClick: write GVL.SwLimitPos via Default
END_VISUALIZATION

// ---- VISUs/COMMAND VISUS/Homing.TcVIS
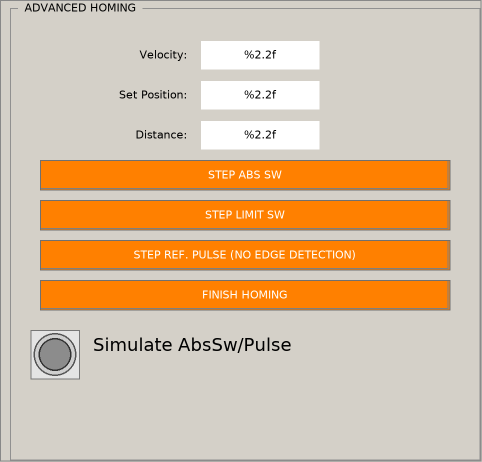
VISUALIZATION Homing  // 482x462
    GroupBox (10,0 470x460), "ADVANCED HOMING"
        Button (30,160 410x30), "STEP ABS SW"
            OnMouseClick: execute { GVL.axes[MAIN.hmiAxisSelect].eCommand:=eMcCommand.HomeStepAbsoluteSwitch; GVL.axes[MAIN.hmiAxisSelect].bEXECUTE:= TRUE; }
        Textfield (190,40 120x30), "%2.2f", text variable: GVL.axes[MAIN.hmiAxisSelect].fHomeVelocity
            OnMouseClick: write GVL.axes[MAIN.hmiAxisSelect].fHomeVelocity via Default
        Textfield (190,80 120x30), "%2.2f", text variable: GVL.axes[MAIN.hmiAxisSelect].fHomePosition
            OnMouseClick: write GVL.axes[MAIN.hmiAxisSelect].fHomePosition via Default
        Textfield (20,40 160x30), "Velocity:"
        Textfield (20,80 160x30), "Set Position:"
        Textfield (20,120 160x30), "Distance:"
        Button (30,280 410x30), "FINISH HOMING"
            OnMouseClick: execute { GVL.axes[MAIN.hmiAxisSelect].eCommand:=eMcCommand.HomeFinish; GVL.axes[MAIN.hmiAxisSelect].bEXECUTE:= TRUE; }
        PushSwitchLed (20,330 50x49), variable: GVL.axes[MAIN.hmiAxisSelect].MCSignalRef.Level, behaviour: TOGGLE, style: Switch-PushSwitchLed-Gray
        Button (30,200 410x30), "STEP LIMIT SW"
            OnMouseClick: execute { GVL.axes[MAIN.hmiAxisSelect].eCommand:=eMcCommand.HomeStepLimitSwitch; GVL.axes[MAIN.hmiAxisSelect].bEXECUTE:= TRUE; }
        Button (30,240 410x30), "STEP REF. PULSE (NO EDGE DETECTION)"
            OnMouseClick: execute { GVL.axes[MAIN.hmiAxisSelect].eCommand:=eMcCommand.HomeStepReferencePulse; GVL.axes[MAIN.hmiAxisSelect].bEXECUTE:= TRUE; }
    Textfield (200,120 120x30), "%2.2f", text variable: GVL.axes[MAIN.hmiAxisSelect].fHomeDistance
        OnMouseClick: write GVL.axes[MAIN.hmiAxisSelect].fHomeDistance via Default
    Label (90,330 280x30), "Simulate AbsSw/Pulse"
END_VISUALIZATION

// ---- VISUs/COMMAND VISUS/AxisSimulation.TcVIS
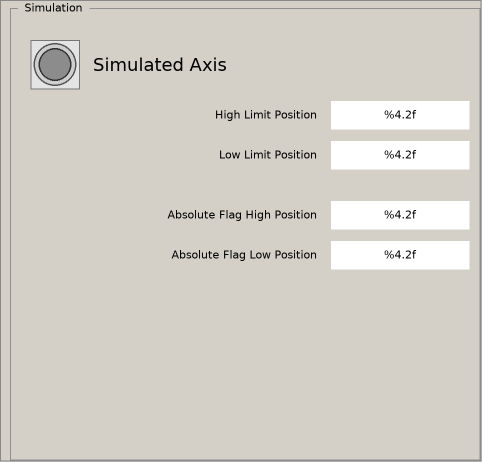
VISUALIZATION AxisSimulation  // 482x462
    GroupBox (10,0 470x460), "Simulation"
        PushSwitchLed (20,40 50x49), variable: MAIN.bSimulate[MAIN.hmiAxisSelect], behaviour: TOGGLE, style: Switch-PushSwitchLed-Gray
        Label (80,50 190x30), "Simulated Axis"
        Textfield (100,100 210x30), "High Limit Position", text variable: MAIN.hmiAxisSelect
        Textfield (320,100 140x30), "%4.2f", text variable: MAIN.simulated[MAIN.hmiAxisSelect].fHighLim
            OnMouseClick: write MAIN.simulated[MAIN.hmiAxisSelect].fHighLim via Default
        Textfield (100,140 210x30), "Low Limit Position", text variable: MAIN.hmiAxisSelect
        Textfield (320,240 140x30), "%4.2f", text variable: MAIN.simulated[MAIN.hmiAxisSelect].fLowAbs
            OnMouseClick: write MAIN.simulated[MAIN.hmiAxisSelect].fLowAbs via Default
    Textfield (330,140 140x30), "%4.2f", text variable: MAIN.simulated[MAIN.hmiAxisSelect].fLowLim
        OnMouseClick: write MAIN.simulated[MAIN.hmiAxisSelect].fLowLim via Default
    Textfield (110,200 210x30), "Absolute Flag High Position", text variable: MAIN.hmiAxisSelect
    Textfield (330,200 140x30), "%4.2f", text variable: MAIN.simulated[MAIN.hmiAxisSelect].fHighAbs
        OnMouseClick: write MAIN.simulated[MAIN.hmiAxisSelect].fHighAbs via Default
    Textfield (110,240 210x30), "Absolute Flag Low Position", text variable: MAIN.hmiAxisSelect
END_VISUALIZATION

// ---- VISUs/Main.TcVIS
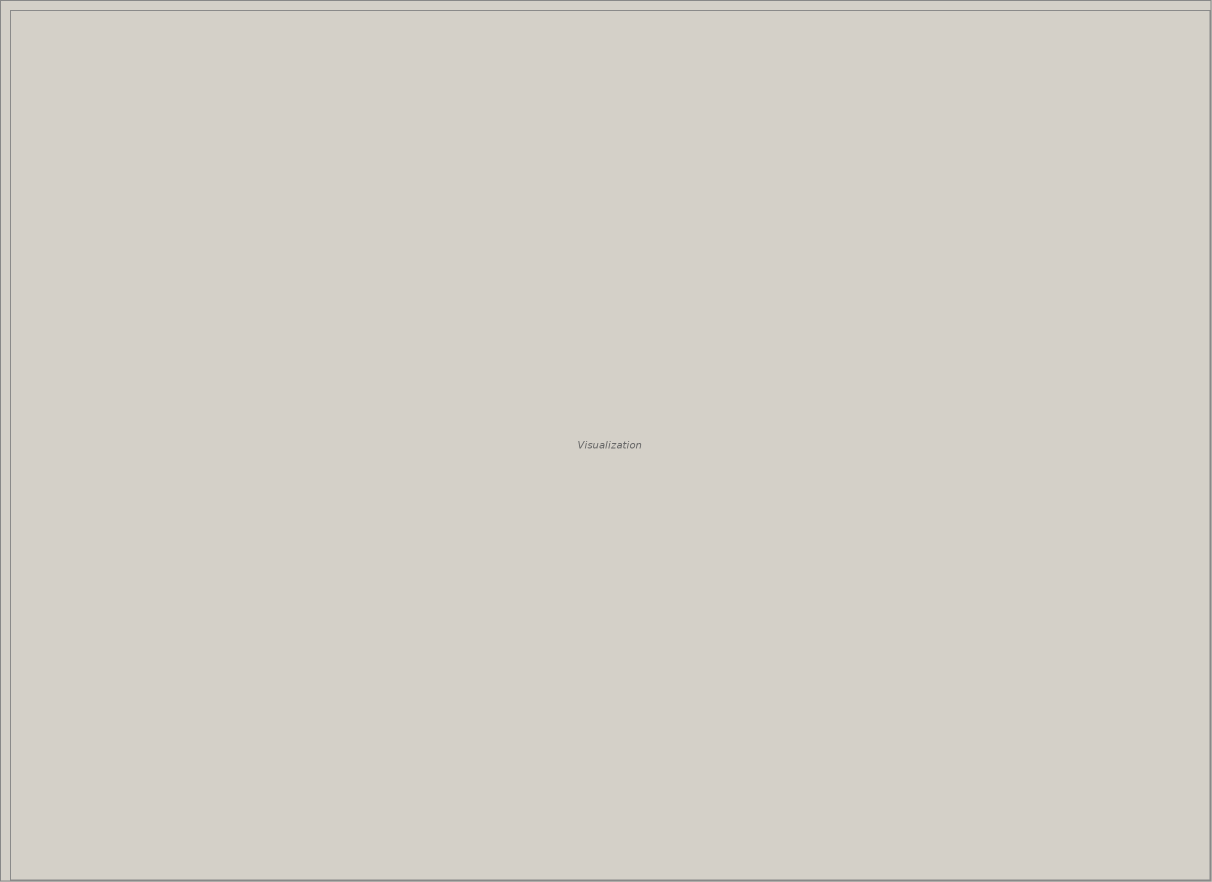
VISUALIZATION Main  // 1212x882
    TabControl (10,10 1200x870)
        shows Visualization()
        shows SlitSet()
        shows IO()
        [0]: TabTitle=Single Axis
        [1]: TabTitle=Slit Set
END_VISUALIZATION

// ---- VISUs/Panels/ButtonStates.TcTLO
TEXTLIST ButtonStates
  0 = 'Enable'
  1 = 'Disable'
   = ''
END_TEXTLIST

// ---- VISUs/Panels/Command VISUs/AxisSimulation.TcVIS
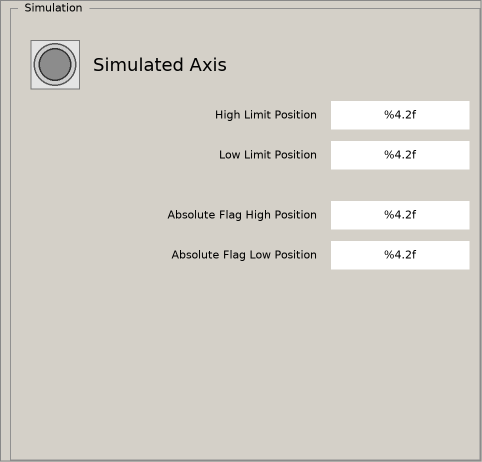
VISUALIZATION AxisSimulation  // 482x462
    GroupBox (10,0 470x460), "Simulation"
        PushSwitchLed (20,40 50x49), variable: MAIN.bSimulate[MAIN.hmiAxisSelect], behaviour: TOGGLE, style: Switch-PushSwitchLed-Gray
        Label (80,50 190x30), "Simulated Axis"
        Textfield (100,100 210x30), "High Limit Position", text variable: MAIN.hmiAxisSelect
        Textfield (320,100 140x30), "%4.2f", text variable: MAIN.simulated[MAIN.hmiAxisSelect].fHighLim
            OnMouseClick: write MAIN.simulated[MAIN.hmiAxisSelect].fHighLim via Default
        Textfield (100,140 210x30), "Low Limit Position", text variable: MAIN.hmiAxisSelect
        Textfield (320,240 140x30), "%4.2f", text variable: MAIN.simulated[MAIN.hmiAxisSelect].fLowAbs
            OnMouseClick: write MAIN.simulated[MAIN.hmiAxisSelect].fLowAbs via Default
    Textfield (330,140 140x30), "%4.2f", text variable: MAIN.simulated[MAIN.hmiAxisSelect].fLowLim
        OnMouseClick: write MAIN.simulated[MAIN.hmiAxisSelect].fLowLim via Default
    Textfield (110,200 210x30), "Absolute Flag High Position", text variable: MAIN.hmiAxisSelect
    Textfield (330,200 140x30), "%4.2f", text variable: MAIN.simulated[MAIN.hmiAxisSelect].fHighAbs
        OnMouseClick: write MAIN.simulated[MAIN.hmiAxisSelect].fHighAbs via Default
    Textfield (110,240 210x30), "Absolute Flag Low Position", text variable: MAIN.hmiAxisSelect
END_VISUALIZATION

// ---- VISUs/Panels/Command VISUs/Gearing.TcVIS
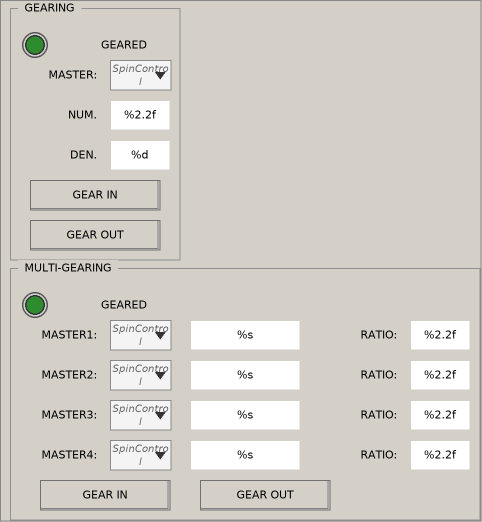
VISUALIZATION Gearing  // 482x522
    GroupBox (10,0 170x260), "GEARING"
        Textfield (40,30 100x30), "GEARED", text variable: MAIN.hmiAxisSelect
        SpinControl (100,60 61x30), variable: GVL.axes[MAIN.hmiAxisSelect].masterAxis
            p651134158: GVL.axisNumMax
            OnMouseClick: write GVL.axes[MAIN.hmiAxisSelect].masterAxis via Default
        Textfield (10,60 80x30), "MASTER:", text variable: MAIN.hmiAxisSelect
        Textfield (100,100 60x30), "%2.2f", text variable: GVL.axes[MAIN.hmiAxisSelect].fGearRatioNum
            OnMouseClick: write GVL.axes[MAIN.hmiAxisSelect].fGearRatioNum via Default
        Textfield (10,100 80x30), "NUM.", text variable: MAIN.hmiAxisSelect
        Textfield (100,140 60x30), "%d", text variable: GVL.axes[MAIN.hmiAxisSelect].iGearRatioDen
            OnMouseClick: write GVL.axes[MAIN.hmiAxisSelect].iGearRatioDen via Default
        Textfield (10,140 80x30), "DEN.", text variable: MAIN.hmiAxisSelect
        Button (20,180 130x30), "GEAR IN"
            OnMouseClick: execute { GVL.axes[MAIN.hmiAxisSelect].eCommand:=eMcCommand.GearIn; GVL.axes[MAIN.hmiAxisSelect].bExecute:= TRUE; }
        Button (20,220 130x30), "GEAR OUT"
            OnMouseClick: execute { GVL.axes[MAIN.hmiAxisSelect].eCommand:=eMcCommand.GearOut; GVL.axes[MAIN.hmiAxisSelect].bExecute:= TRUE; }
        Lamp1 (10,30 30x30), variable: GVL.axes[MAIN.hmiAxisSelect].iAxisState=500, style: Lamp-Lamp1-Green
    GroupBox (10,260 470x260), "MULTI-GEARING"
        Lamp1 (10,30 30x30), variable: GVL.axes[MAIN.hmiAxisSelect].iAxisState=500, style: Lamp-Lamp1-Green
        Textfield (40,30 100x30), "GEARED", text variable: MAIN.hmiAxisSelect
        SpinControl (100,60 61x30), variable: GVL.axes[MAIN.hmiAxisSelect].masterAxes[1].i
            p651134158: GVL.axisNumMax
            OnMouseClick: write GVL.axes[MAIN.hmiAxisSelect].masterAxes[1].i via Default
        Textfield (10,60 80x30), "MASTER1:", text variable: MAIN.hmiAxisSelect
        Textfield (400,60 60x30), "%2.2f", text variable: GVL.axes[MAIN.hmiAxisSelect].masterAxes[1].ratio
            OnMouseClick: write GVL.axes[MAIN.hmiAxisSelect].masterAxes[1].ratio via Default
        Textfield (310,60 80x30), "RATIO:", text variable: MAIN.hmiAxisSelect
        Button (30,220 130x30), "GEAR IN"
            OnMouseClick: execute { GVL.axes[MAIN.hmiAxisSelect].eCommand:=eMcCommand.GearInMultiMaster; GVL.axes[MAIN.hmiAxisSelect].bExecute:= TRUE; }
        Button (190,220 130x30), "GEAR OUT"
            OnMouseClick: execute { GVL.axes[MAIN.hmiAxisSelect].eCommand:=eMcCommand.GearOut; GVL.axes[MAIN.hmiAxisSelect].bExecute:= TRUE; }
        SpinControl (100,100 61x30), variable: GVL.axes[MAIN.hmiAxisSelect].masterAxes[2].i
            p651134158: GVL.axisNumMax
            OnMouseClick: write GVL.axes[MAIN.hmiAxisSelect].masterAxes[2].i via Default
        SpinControl (100,140 61x30), variable: GVL.axes[MAIN.hmiAxisSelect].masterAxes[3].i
            p651134158: GVL.axisNumMax
            OnMouseClick: write GVL.axes[MAIN.hmiAxisSelect].masterAxes[3].i via Default
        SpinControl (100,180 61x30), variable: GVL.axes[MAIN.hmiAxisSelect].masterAxes[4].i
            p651134158: GVL.axisNumMax
            OnMouseClick: write GVL.axes[MAIN.hmiAxisSelect].masterAxes[4].i via Default
        Textfield (310,100 80x30), "RATIO:", text variable: MAIN.hmiAxisSelect
        Textfield (310,140 80x30), "RATIO:", text variable: MAIN.hmiAxisSelect
        Textfield (310,180 80x30), "RATIO:", text variable: MAIN.hmiAxisSelect
        Textfield (10,100 80x30), "MASTER2:", text variable: MAIN.hmiAxisSelect
        Textfield (10,140 80x30), "MASTER3:", text variable: MAIN.hmiAxisSelect
        Textfield (10,180 80x30), "MASTER4:", text variable: MAIN.hmiAxisSelect
        Textfield (400,100 60x30), "%2.2f", text variable: GVL.axes[MAIN.hmiAxisSelect].masterAxes[2].ratio
            OnMouseClick: write GVL.axes[MAIN.hmiAxisSelect].masterAxes[2].ratio via Default
        Textfield (400,140 60x30), "%2.2f", text variable: GVL.axes[MAIN.hmiAxisSelect].masterAxes[3].ratio
            OnMouseClick: write GVL.axes[MAIN.hmiAxisSelect].masterAxes[3].ratio via Default
        Textfield (400,180 60x30), "%2.2f", text variable: GVL.axes[MAIN.hmiAxisSelect].masterAxes[4].ratio
            OnMouseClick: write GVL.axes[MAIN.hmiAxisSelect].masterAxes[4].ratio via Default
        Textfield (180,60 110x30), "%s", text variable: GVL.axes[GVL.axes[MAIN.hmiAxisSelect].masterAxes[1].i].sAxisName
        Textfield (180,100 110x30), "%s", text variable: GVL.axes[GVL.axes[MAIN.hmiAxisSelect].masterAxes[2].i].sAxisName
        Textfield (180,140 110x30), "%s", text variable: GVL.axes[GVL.axes[MAIN.hmiAxisSelect].masterAxes[3].i].sAxisName
        Textfield (180,180 110x30), "%s", text variable: GVL.axes[GVL.axes[MAIN.hmiAxisSelect].masterAxes[4].i].sAxisName
END_VISUALIZATION

// ---- VISUs/Panels/Command VISUs/Homing.TcVIS
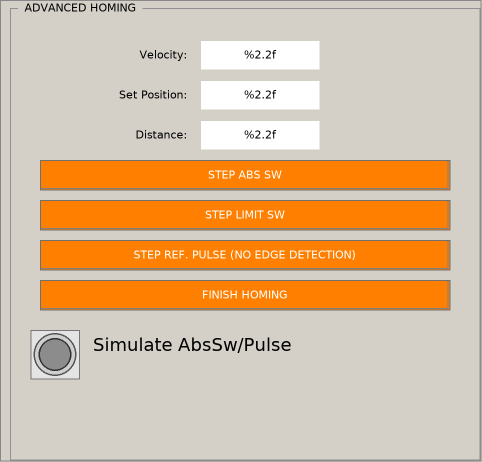
VISUALIZATION Homing  // 482x462
    GroupBox (10,0 470x460), "ADVANCED HOMING"
        Button (30,160 410x30), "STEP ABS SW"
            OnMouseClick: execute { GVL.axes[MAIN.hmiAxisSelect].eCommand:=eMcCommand.HomeStepAbsoluteSwitch; GVL.axes[MAIN.hmiAxisSelect].bEXECUTE:= TRUE; }
        Textfield (190,40 120x30), "%2.2f", text variable: GVL.axes[MAIN.hmiAxisSelect].fHomeVelocity
            OnMouseClick: write GVL.axes[MAIN.hmiAxisSelect].fHomeVelocity via Default
        Textfield (190,80 120x30), "%2.2f", text variable: GVL.axes[MAIN.hmiAxisSelect].fHomePosition
            OnMouseClick: write GVL.axes[MAIN.hmiAxisSelect].fHomePosition via Default
        Textfield (20,40 160x30), "Velocity:"
        Textfield (20,80 160x30), "Set Position:"
        Textfield (20,120 160x30), "Distance:"
        Button (30,280 410x30), "FINISH HOMING"
            OnMouseClick: execute { GVL.axes[MAIN.hmiAxisSelect].eCommand:=eMcCommand.HomeFinish; GVL.axes[MAIN.hmiAxisSelect].bEXECUTE:= TRUE; }
        PushSwitchLed (20,330 50x49), variable: GVL.axes[MAIN.hmiAxisSelect].MCSignalRef.Level, behaviour: TOGGLE, style: Switch-PushSwitchLed-Gray
        Button (30,200 410x30), "STEP LIMIT SW"
            OnMouseClick: execute { GVL.axes[MAIN.hmiAxisSelect].eCommand:=eMcCommand.HomeStepLimitSwitch; GVL.axes[MAIN.hmiAxisSelect].bEXECUTE:= TRUE; }
        Button (30,240 410x30), "STEP REF. PULSE (NO EDGE DETECTION)"
            OnMouseClick: execute { GVL.axes[MAIN.hmiAxisSelect].eCommand:=eMcCommand.HomeStepReferencePulse; GVL.axes[MAIN.hmiAxisSelect].bEXECUTE:= TRUE; }
    Textfield (200,120 120x30), "%2.2f", text variable: GVL.axes[MAIN.hmiAxisSelect].fHomeDistance
        OnMouseClick: write GVL.axes[MAIN.hmiAxisSelect].fHomeDistance via Default
    Label (90,330 280x30), "Simulate AbsSw/Pulse"
END_VISUALIZATION

// ---- VISUs/Panels/Command VISUs/Parameters.TcVIS
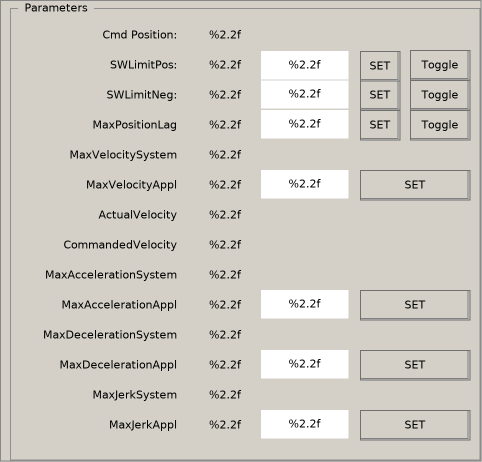
VISUALIZATION Parameters  // 482x462
    GroupBox (10,0 470x460), "Parameters"
        Textfield (170,20 90x30), "%2.2f", text variable: GVL.axes[MAIN.hmiAxisSelect].fParameters[1]
        Textfield (10,50 160x30), "SWLimitPos:"
        Textfield (10,20 160x30), "Cmd Position:"
        Textfield (170,50 90x30), "%2.2f", text variable: GVL.axes[MAIN.hmiAxisSelect].fParameters[2], input disabled if: NOT GVL.axes[MAIN.hmiAxisSelect].bSoftLimPosEn
        Textfield (170,80 90x30), "%2.2f", text variable: GVL.axes[MAIN.hmiAxisSelect].fParameters[3], input disabled if: NOT GVL.axes[MAIN.hmiAxisSelect].bSoftLimNegEn
        Textfield (250,79 89x30), "%2.2f", text variable: GVL.SwLimitNeg
            OnMouseClick: write GVL.SwLimitNeg via Default
        Button (350,80 40x30), "SET"
            toggle GVL.axes[MAIN.hmiAxisSelect].bEXECUTE
            OnMouseClick: execute {
                GVL.axes[Main.hmiAxisSelect].eCommand:=eMcCommand.WriteParameter;
                GVL.axes[Main.hmiAxisSelect].fParameterValue:=GVL.SwLimitNeg;
                GVL.axes[Main.hmiAxisSelect].iParameterIndex:=eRWParameter.SWLimitNeg;
                GVL.axes[Main.hmiAxisSelect].bExecute:=TRUE;
            }
        Button (400,50 60x30), "Toggle", pressed state: GVL.axes[MAIN.hmiAxisSelect].bSoftLimPosEn, text list: 'ButtonStates', text index: GVL.axes[MAIN.hmiAxisSelect].bSoftLimPosEn
            toggle GVL.axes[MAIN.hmiAxisSelect].bEXECUTE
            OnMouseClick: execute {
                GVL.axes[MAIN.hmiAxisSelect].bInput:=NOT GVL.axes[MAIN.hmiAxisSelect].bSoftLimPosEn;
                GVL.axes[MAIN.hmiAxisSelect].eCommand:=eMcCommand.WriteBoolParameter;
                GVL.axes[MAIN.hmiAxisSelect].iParameterIndex:=eRWParameter.EnableLimitPos;
                GVL.axes[MAIN.hmiAxisSelect].bExecute:=TRUE;
            }
        Button (400,80 60x30), "Toggle", pressed state: GVL.axes[MAIN.hmiAxisSelect].bSoftLimNegEn, text list: 'ButtonStates', text index: GVL.axes[MAIN.hmiAxisSelect].bSoftLimNegEn
            toggle GVL.axes[MAIN.hmiAxisSelect].bEXECUTE
            OnMouseClick: execute {
                GVL.axes[MAIN.hmiAxisSelect].bInput:=NOT GVL.axes[MAIN.hmiAxisSelect].bSoftLimNegEn;
                GVL.axes[MAIN.hmiAxisSelect].eCommand:=eMcCommand.WriteBoolParameter;
                GVL.axes[MAIN.hmiAxisSelect].iParameterIndex:=eRWParameter.EnableLimitNeg;
                GVL.axes[MAIN.hmiAxisSelect].bExecute:=TRUE;
            }
        Textfield (10,110 160x30), "MaxPositionLag"
        Textfield (10,140 160x30), "MaxVelocitySystem"
        Textfield (10,170 160x30), "MaxVelocityAppl"
        Textfield (10,200 160x30), "ActualVelocity"
        Textfield (10,230 160x30), "CommandedVelocity"
        Textfield (170,260 90x30), "%2.2f", text variable: GVL.axes[MAIN.hmiAxisSelect].fParameters[12]
        Textfield (10,290 160x30), "MaxAccelerationAppl"
        Textfield (10,320 160x30), "MaxDecelerationSystem"
        Textfield (10,380 160x30), "MaxJerkSystem"
        Button (350,51 40x30), "SET"
            toggle GVL.axes[MAIN.hmiAxisSelect].bEXECUTE
            OnMouseClick: execute {
                GVL.axes[Main.hmiAxisSelect].eCommand:=eMcCommand.WriteParameter;
                GVL.axes[Main.hmiAxisSelect].fParameterValue:=GVL.SwLimitPos;
                GVL.axes[Main.hmiAxisSelect].iParameterIndex:=eRWParameter.SWLimitPos;
                GVL.axes[Main.hmiAxisSelect].bExecute:=TRUE;
            }
        Textfield (10,80 160x30), "SWLimitNeg:"
        Textfield (170,110 90x30), "%2.2f", text variable: GVL.axes[MAIN.hmiAxisSelect].fParameters[7], input disabled if: NOT GVL.axes[MAIN.hmiAxisSelect].bPosLagEn
        Textfield (250,109 89x30), "%2.2f", text variable: GVL.MaxPositionLag
            OnMouseClick: write GVL.MaxPositionLag via Default
        Button (350,110 40x30), "SET"
            toggle GVL.axes[MAIN.hmiAxisSelect].bEXECUTE
            OnMouseClick: execute {
                GVL.axes[Main.hmiAxisSelect].eCommand:=eMcCommand.WriteParameter;
                GVL.axes[Main.hmiAxisSelect].fParameterValue:=GVL.MaxPositionLag;
                GVL.axes[Main.hmiAxisSelect].iParameterIndex:=eRWParameter.MaxPositionLag;
                GVL.axes[Main.hmiAxisSelect].bExecute:=TRUE;
            }
        Button (400,110 60x30), "Toggle", pressed state: GVL.axes[MAIN.hmiAxisSelect].bPosLagEn, text list: 'ButtonStates', text index: GVL.axes[MAIN.hmiAxisSelect].bPosLagEn
            toggle GVL.axes[MAIN.hmiAxisSelect].bEXECUTE
            OnMouseClick: execute {
                GVL.axes[MAIN.hmiAxisSelect].bInput:=NOT GVL.axes[MAIN.hmiAxisSelect].bPosLagEn;
                GVL.axes[MAIN.hmiAxisSelect].eCommand:=eMcCommand.WriteBoolParameter;
                GVL.axes[MAIN.hmiAxisSelect].iParameterIndex:=eRWParameter.EnablePosLagMonitoring;
                GVL.axes[MAIN.hmiAxisSelect].bExecute:=TRUE;
            }
        Textfield (170,140 90x30), "%2.2f", text variable: GVL.axes[MAIN.hmiAxisSelect].fParameters[8]
        Textfield (170,170 90x30), "%2.2f", text variable: GVL.axes[MAIN.hmiAxisSelect].fParameters[9]
        Textfield (250,169 89x30), "%2.2f", text variable: GVL.MaxVelocityAppl
            OnMouseClick: write GVL.MaxVelocityAppl via Default
        Button (350,170 110x30), "SET"
            toggle GVL.axes[MAIN.hmiAxisSelect].bEXECUTE
            OnMouseClick: execute {
                GVL.axes[Main.hmiAxisSelect].eCommand:=eMcCommand.WriteParameter;
                GVL.axes[Main.hmiAxisSelect].fParameterValue:=GVL.MaxVelocityAppl;
                GVL.axes[Main.hmiAxisSelect].iParameterIndex:=eRWParameter.MaxVelocityAppl;
                GVL.axes[Main.hmiAxisSelect].bExecute:=TRUE;
            }
        Textfield (170,200 90x30), "%2.2f", text variable: GVL.axes[MAIN.hmiAxisSelect].fParameters[10]
        Textfield (170,230 90x30), "%2.2f", text variable: GVL.axes[MAIN.hmiAxisSelect].fParameters[11]
        Textfield (10,260 160x30), "MaxAccelerationSystem"
        Textfield (170,290 90x30), "%2.2f", text variable: GVL.axes[MAIN.hmiAxisSelect].fParameters[13]
        Textfield (250,289 89x30), "%2.2f", text variable: GVL.MaxAccelerationAppl
            OnMouseClick: write GVL.MaxAccelerationAppl via Default
        Button (350,290 110x30), "SET"
            toggle GVL.axes[MAIN.hmiAxisSelect].bEXECUTE
            OnMouseClick: execute {
                GVL.axes[Main.hmiAxisSelect].eCommand:=eMcCommand.WriteParameter;
                GVL.axes[Main.hmiAxisSelect].fParameterValue:=GVL.MaxAccelerationAppl;
                GVL.axes[Main.hmiAxisSelect].iParameterIndex:=eRWParameter.MaxAccelerationAppl;
                GVL.axes[Main.hmiAxisSelect].bExecute:=TRUE;
            }
        Textfield (170,320 90x30), "%2.2f", text variable: GVL.axes[MAIN.hmiAxisSelect].fParameters[14]
        Textfield (10,350 160x30), "MaxDecelerationAppl"
        Textfield (170,350 90x30), "%2.2f", text variable: GVL.axes[MAIN.hmiAxisSelect].fParameters[15]
        Textfield (250,349 89x30), "%2.2f", text variable: GVL.MaxDecelerationAppl
            OnMouseClick: write GVL.MaxDecelerationAppl via Default
        Button (350,350 110x30), "SET"
            toggle GVL.axes[MAIN.hmiAxisSelect].bEXECUTE
            OnMouseClick: execute {
                GVL.axes[Main.hmiAxisSelect].eCommand:=eMcCommand.WriteParameter;
                GVL.axes[Main.hmiAxisSelect].fParameterValue:=GVL.MaxDecelerationAppl;
                GVL.axes[Main.hmiAxisSelect].iParameterIndex:=eRWParameter.MaxDecelerationAppl;
                GVL.axes[Main.hmiAxisSelect].bExecute:=TRUE;
            }
        Textfield (170,380 90x30), "%2.2f", text variable: GVL.axes[MAIN.hmiAxisSelect].fParameters[16]
        Textfield (10,410 160x30), "MaxJerkAppl"
        Textfield (170,410 90x30), "%2.2f", text variable: GVL.axes[MAIN.hmiAxisSelect].fParameters[17]
        Textfield (250,409 89x30), "%2.2f", text variable: GVL.MaxJerkAppl
            OnMouseClick: write GVL.MaxJerkAppl via Default
        Button (350,410 110x30), "SET"
            toggle GVL.axes[MAIN.hmiAxisSelect].bEXECUTE
            OnMouseClick: execute {
                GVL.axes[Main.hmiAxisSelect].eCommand:=eMcCommand.WriteParameter;
                GVL.axes[Main.hmiAxisSelect].fParameterValue:=GVL.MaxJerkAppl;
                GVL.axes[Main.hmiAxisSelect].iParameterIndex:=eRWParameter.MaxJerkAppl;
                GVL.axes[Main.hmiAxisSelect].bExecute:=TRUE;
            }
        Textfield (250,50 89x30), "%2.2f", text variable: GVL.SwLimitPos
            OnMouseClick: write GVL.SwLimitPos via Default
END_VISUALIZATION

// ---- VISUs/Panels/CommandList.TcTLO
TEXTLIST CommandList
  1 = 'Reset'
  2 = 'Power'
  3 = 'Read Status'
  4 = 'Read Axis Error'
  5 = 'Read Parameter'
  6 = 'Read Bool Parameter'
  7 = 'Write Parameter'
  8 = 'Write Bool Parameter'
  9 = 'Read Digital Input *'
  10 = 'Read Digital Output*'
  11 = 'Write Digital Output*'
  12 = 'Read Actual Position'
  13 = 'Read Actual Velocity'
  14 = 'Read Actual Torque*'
  15 = 'Read Axis Info*'
  16 = 'Read Motion State *'
  17 = 'Set Position'
  18 = 'Set Override'
  19 = 'Touch Probe'
  20 = 'Digital Cam Switch *'
  21 = 'Abort Trigger'
  22 = 'Abort Superposition'
  23 = 'Cam Table Select'
  24 = 'Home'
  25 = 'Jog'
  26 = 'Stop'
  27 = 'Halt'
  28 = 'Move Absolute'
  29 = 'Move Relative'
  30 = 'Move Additive'
  31 = 'Move Superimposed'
  32 = 'Move Velocity'
  33 = 'Move Continuous Absolute'
  34 = 'Move Continuous Relative'
  35 = 'Move Modulo'
  36 = 'Torque Control *'
  37 = 'Position Profile *'
  38 = 'Velocity Profile *'
  39 = 'Acceleration Profile *'
  40 = 'Gear In'
  41 = 'Gear In Dynamic'
  42 = 'Gear In Multi-Master'
  43 = 'Gear Out'
  44 = 'Halt Phasing'
  45 = 'Phasing Absolute'
  46 = 'Phasing Relative'
  47 = 'Cam In'
  48 = 'Cam Out'
  49 = 'Cam Scaling'
  50 = 'Cam Add'
  51 = 'Cam Exchange'
  52 = 'Cam In V2'
  53 = 'Cam Remove'
  54 = 'Cam Scaling V2'
   = ''
END_TEXTLIST

// ---- VISUs/Panels/IO.TcVIS
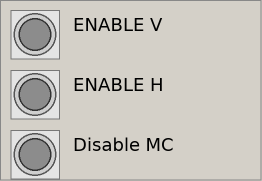
VISUALIZATION IO  // 262x181
    PushSwitchLed (10,10 50x49), variable: MAIN.limitEnable1, behaviour: TOGGLE, style: Switch-PushSwitchLed-Gray
    PushSwitchLed (10,70 50x49), variable: MAIN.limitEnable2, behaviour: TOGGLE, style: Switch-PushSwitchLed-Gray
    Label (70,10 190x30), "ENABLE V"
    Label (70,70 190x30), "ENABLE H"
    PushSwitchLed (10,130 50x49), variable: MAIN.bDisableMC, behaviour: TOGGLE, style: Switch-PushSwitchLed-Gray
    Label (70,130 190x30), "Disable MC"
END_VISUALIZATION

// ---- VISUs/Panels/SlitSet.TcVIS
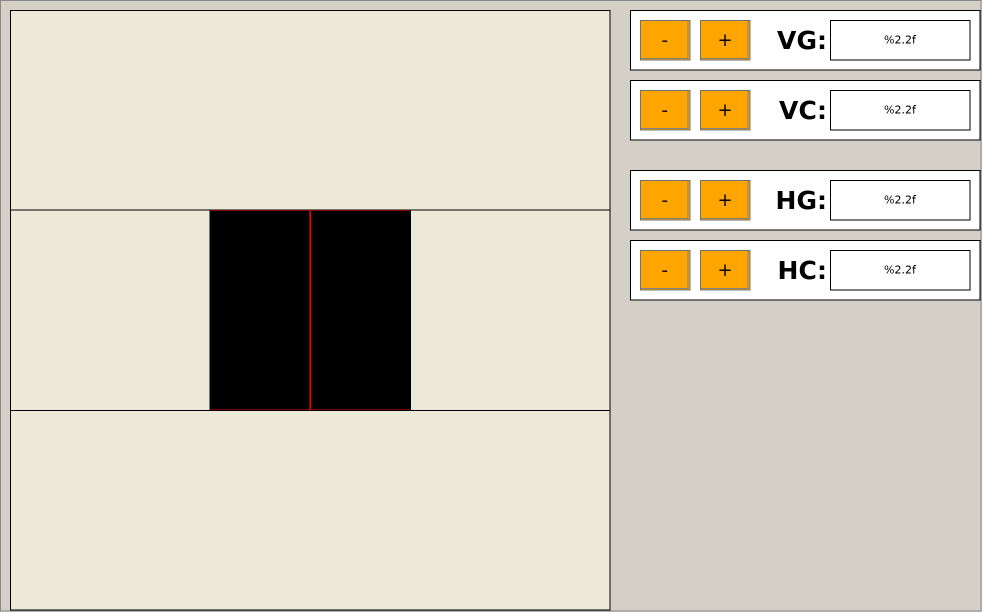
VISUALIZATION SlitSet  // 982x612
    Rectangle (630,10 350x60)
    Rectangle (210,210 200x200)
    Rectangle (210,160 200x150)
        p2738717112: -GVL.axes[1].Axis.NcToPlc.ActPos
    Rectangle (210,310 200x150)
        p2738717112: -GVL.axes[2].Axis.NcToPlc.ActPos
    Rectangle (310,210 150x200)
        p3560616238: GVL.axes[3].Axis.NcToPlc.ActPos
    Rectangle (160,210 150x200)
        p3560616238: GVL.axes[4].Axis.NcToPlc.ActPos
    Rectangle (410,160 200x300)
    Rectangle (10,160 200x300)
    Rectangle (10,10 600x200)
    Rectangle (10,410 600x200)
    Textfield (830,20 140x40), "%2.2f", text variable: GVL.axes[5].Axis.NcToPlc.ActPos
    Button (700,20 50x40), "+"
        tap GVL.axes[5].bJogForward
        OnMouseClick: execute { GVL.axes[5].eCommand:=eMcCommand.Jog; }
    Button (640,20 50x40), "-"
        tap GVL.axes[5].bJogBackward
        OnMouseClick: execute { GVL.axes[5].eCommand:=eMcCommand.Jog; }
    Textfield (760,20 70x40), "VG:"
    Rectangle (630,80 350x60)
    Textfield (830,90 140x40), "%2.2f", text variable: GVL.axes[6].Axis.NcToPlc.ActPos
    Button (700,90 50x40), "+"
        tap GVL.axes[6].bJogForward
        OnMouseClick: execute { GVL.axes[6].eCommand:=eMcCommand.Jog; }
    Button (640,90 50x40), "-"
        tap GVL.axes[6].bJogBackward
        OnMouseClick: execute { GVL.axes[6].eCommand:=eMcCommand.Jog; }
    Textfield (760,90 70x40), "VC:"
    Rectangle (630,170 350x60)
    Textfield (830,180 140x40), "%2.2f", text variable: GVL.axes[7].Axis.NcToPlc.ActPos
    Button (700,180 50x40), "+"
        tap GVL.axes[7].bJogForward
        OnMouseClick: execute { GVL.axes[7].eCommand:=eMcCommand.Jog; }
    Button (640,180 50x40), "-"
        tap GVL.axes[7].bJogBackward
        OnMouseClick: execute { GVL.axes[7].eCommand:=eMcCommand.Jog; }
    Textfield (760,180 70x40), "HG:"
    Rectangle (630,240 350x60)
    Textfield (830,250 140x40), "%2.2f", text variable: GVL.axes[8].Axis.NcToPlc.ActPos
    Button (700,250 50x40), "+"
        tap GVL.axes[8].bJogForward
        OnMouseClick: execute { GVL.axes[8].eCommand:=eMcCommand.Jog; }
    Button (640,250 50x40), "-"
        tap GVL.axes[8].bJogBackward
        OnMouseClick: execute { GVL.axes[8].eCommand:=eMcCommand.Jog; }
    Textfield (760,250 70x40), "HC:"
END_VISUALIZATION

